//     PlcTask Outputs/GVL_iXlinker.EtherCAT_Master_ATxxxx.Beckhoff_AT1xxx.Beckhoff_AT2xxxEK1122.A_0023_AT2002_0250_0022.CC_Outputs.Control <-> CC Outputs/Control
//     PlcTask Outputs/GVL_iXlinker.EtherCAT_Master_ATxxxx.Beckhoff_AT1xxx.Beckhoff_AT2xxxEK1122.A_0023_AT2002_0250_0022.CC_Outputs.Current_setpoint_value_Ch[0] <-> CC Outputs/Current setpoint value Ch.1
//     PlcTask Outputs/GVL_iXlinker.EtherCAT_Master_ATxxxx.Beckhoff_AT1xxx.Beckhoff_AT2xxxEK1122.A_0023_AT2002_0250_0022.CC_Outputs.Current_setpoint_value_Ch[1] <-> CC Outputs/Current setpoint value Ch.2
//     PlcTask Outputs/GVL_iXlinker.EtherCAT_Master_ATxxxx.Beckhoff_AT1xxx.Beckhoff_AT2xxxEK1122.A_0023_AT2002_0250_0022.CC_Outputs.Current_setpoint_value_Ch[2] <-> CC Outputs/Current setpoint value Ch.3
//     PlcTask Outputs/GVL_iXlinker.EtherCAT_Master_ATxxxx.Beckhoff_AT1xxx.Beckhoff_AT2xxxEK1122.A_0023_AT2002_0250_0022.CC_Outputs.Current_setpoint_value_Ch[3] <-> CC Outputs/Current setpoint value Ch.4
//     PlcTask Outputs/GVL_iXlinker.EtherCAT_Master_ATxxxx.Beckhoff_AT1xxx.Beckhoff_AT2xxxEK1122.A_0023_AT2002_0250_0022.CC_Outputs.Current_setpoint_value_Ch[4] <-> CC Outputs/Current setpoint value Ch.5
//     PlcTask Outputs/GVL_iXlinker.EtherCAT_Master_ATxxxx.Beckhoff_AT1xxx.Beckhoff_AT2xxxEK1122.A_0023_AT2002_0250_0022.CC_Outputs.Current_setpoint_value_Ch[5] <-> CC Outputs/Current setpoint value Ch.6
//     PlcTask Outputs/GVL_iXlinker.EtherCAT_Master_ATxxxx.Beckhoff_AT1xxx.Beckhoff_AT2xxxEK1122.A_0023_AT2002_0250_0022.CC_Outputs.Current_setpoint_value_Ch[6] <-> CC Outputs/Current setpoint value Ch.7
//     PlcTask Outputs/GVL_iXlinker.EtherCAT_Master_ATxxxx.Beckhoff_AT1xxx.Beckhoff_AT2xxxEK1122.A_0023_AT2002_0250_0022.CC_Outputs.Current_setpoint_value_Ch[7] <-> CC Outputs/Current setpoint value Ch.8
//     PlcTask Outputs/GVL_iXlinker.EtherCAT_Master_ATxxxx.Beckhoff_AT1xxx.Beckhoff_AT2xxxEK1122.A_0023_AT2002_0250_0022.CC_Outputs.Current_setpoint_value_Ch[8] <-> CC Outputs/Current setpoint value Ch.9
//     PlcTask Outputs/GVL_iXlinker.EtherCAT_Master_ATxxxx.Beckhoff_AT1xxx.Beckhoff_AT2xxxEK1122.A_0023_AT2002_0250_0022.CC_Outputs.Current_setpoint_value_Ch[9] <-> CC Outputs/Current setpoint value Ch.10
//     PlcTask Outputs/GVL_iXlinker.EtherCAT_Master_ATxxxx.Beckhoff_AT1xxx.Beckhoff_AT2xxxEK1122.A_0023_AT2002_0250_0022.CC_Outputs.Current_setpoint_value_Ch[10] <-> CC Outputs/Current setpoint value Ch.11
//     PlcTask Outputs/GVL_iXlinker.EtherCAT_Master_ATxxxx.Beckhoff_AT1xxx.Beckhoff_AT2xxxEK1122.A_0023_AT2002_0250_0022.CC_Outputs.Current_setpoint_value_Ch[11] <-> CC Outputs/Current setpoint value Ch.12
//     PlcTask Outputs/GVL_iXlinker.EtherCAT_Master_ATxxxx.Beckhoff_AT1xxx.Beckhoff_AT2xxxEK1122.A_0023_AT2002_0250_0022.CC_Outputs.Current_setpoint_value_Ch[12] <-> CC Outputs/Current setpoint value Ch.13
//     PlcTask Outputs/GVL_iXlinker.EtherCAT_Master_ATxxxx.Beckhoff_AT1xxx.Beckhoff_AT2xxxEK1122.A_0023_AT2002_0250_0022.CC_Outputs.Current_setpoint_value_Ch[13] <-> CC Outputs/Current setpoint value Ch.14
//     PlcTask Outputs/GVL_iXlinker.EtherCAT_Master_ATxxxx.Beckhoff_AT1xxx.Beckhoff_AT2xxxEK1122.A_0023_AT2002_0250_0022.CC_Outputs.Current_setpoint_value_Ch[14] <-> CC Outputs/Current setpoint value Ch.15
//     PlcTask Inputs/GVL_iXlinker.EtherCAT_Master_ATxxxx.Beckhoff_AT1xxx.Beckhoff_AT2xxxEK1122.A_0023_AT2002_0250_0022.WcState.WcState <-> WcState/WcState
//     PlcTask Inputs/GVL_iXlinker.EtherCAT_Master_ATxxxx.Beckhoff_AT1xxx.Beckhoff_AT2xxxEK1122.A_0023_AT2002_0250_0022.WcState.InputToggle <-> WcState/InputToggle
//     PlcTask Inputs/GVL_iXlinker.EtherCAT_Master_ATxxxx.Beckhoff_AT1xxx.Beckhoff_AT2xxxEK1122.A_0023_AT2002_0250_0022.InfoData.AdsAddr <-> InfoData/AdsAddr
//     PlcTask Inputs/GVL_iXlinker.EtherCAT_Master_ATxxxx.Beckhoff_AT1xxx.Beckhoff_AT2xxxEK1122.A_0023_AT2002_0250_0022.InfoData.DcOutputShift <-> InfoData/DcOutputShift
//     PlcTask Inputs/GVL_iXlinker.EtherCAT_Master_ATxxxx.Beckhoff_AT1xxx.Beckhoff_AT2xxxEK1122.A_0023_AT2002_0250_0022.InfoData.DcInputShift <-> InfoData/DcInputShift
//     PlcTask Inputs/GVL_iXlinker.EtherCAT_Master_ATxxxx.Beckhoff_AT1xxx.Beckhoff_AT2xxxEK1122.A_0023_AT2002_0250_0022.InfoData.State <-> InfoData/State
//   PLC/PLC Instance <-> EtherCAT Master ATxxxx/Beckhoff AT1xxx/Beckhoff AT2xxxEK1122/A_0024(AT2002-0250-0023)
//     PlcTask Inputs/GVL_iXlinker.EtherCAT_Master_ATxxxx.Beckhoff_AT1xxx.Beckhoff_AT2xxxEK1122.A_0024_AT2002_0250_0023.CC_Inputs.Status <-> CC Inputs/Status
//     PlcTask Inputs/GVL_iXlinker.EtherCAT_Master_ATxxxx.Beckhoff_AT1xxx.Beckhoff_AT2xxxEK1122.A_0024_AT2002_0250_0023.CC_Inputs.Current_actual_value_Ch[0] <-> CC Inputs/Current actual value Ch.1
//     PlcTask Inputs/GVL_iXlinker.EtherCAT_Master_ATxxxx.Beckhoff_AT1xxx.Beckhoff_AT2xxxEK1122.A_0024_AT2002_0250_0023.CC_Inputs.Current_actual_value_Ch[1] <-> CC Inputs/Current actual value Ch.2
//     PlcTask Inputs/GVL_iXlinker.EtherCAT_Master_ATxxxx.Beckhoff_AT1xxx.Beckhoff_AT2xxxEK1122.A_0024_AT2002_0250_0023.CC_Inputs.Current_actual_value_Ch[2] <-> CC Inputs/Current actual value Ch.3
//     PlcTask Inputs/GVL_iXlinker.EtherCAT_Master_ATxxxx.Beckhoff_AT1xxx.Beckhoff_AT2xxxEK1122.A_0024_AT2002_0250_0023.CC_Inputs.Current_actual_value_Ch[3] <-> CC Inputs/Current actual value Ch.4
//     PlcTask Inputs/GVL_iXlinker.EtherCAT_Master_ATxxxx.Beckhoff_AT1xxx.Beckhoff_AT2xxxEK1122.A_0024_AT2002_0250_0023.CC_Inputs.Current_actual_value_Ch[4] <-> CC Inputs/Current actual value Ch.5
//     PlcTask Inputs/GVL_iXlinker.EtherCAT_Master_ATxxxx.Beckhoff_AT1xxx.Beckhoff_AT2xxxEK1122.A_0024_AT2002_0250_0023.CC_Inputs.Current_actual_value_Ch[5] <-> CC Inputs/Current actual value Ch.6
//     PlcTask Inputs/GVL_iXlinker.EtherCAT_Master_ATxxxx.Beckhoff_AT1xxx.Beckhoff_AT2xxxEK1122.A_0024_AT2002_0250_0023.CC_Inputs.Current_actual_value_Ch[6] <-> CC Inputs/Current actual value Ch.7
//     PlcTask Inputs/GVL_iXlinker.EtherCAT_Master_ATxxxx.Beckhoff_AT1xxx.Beckhoff_AT2xxxEK1122.A_0024_AT2002_0250_0023.CC_Inputs.Current_actual_value_Ch[7] <-> CC Inputs/Current actual value Ch.8
//     PlcTask Inputs/GVL_iXlinker.EtherCAT_Master_ATxxxx.Beckhoff_AT1xxx.Beckhoff_AT2xxxEK1122.A_0024_AT2002_0250_0023.CC_Inputs.Current_actual_value_Ch[8] <-> CC Inputs/Current actual value Ch.9
//     PlcTask Inputs/GVL_iXlinker.EtherCAT_Master_ATxxxx.Beckhoff_AT1xxx.Beckhoff_AT2xxxEK1122.A_0024_AT2002_0250_0023.CC_Inputs.Current_actual_value_Ch[9] <-> CC Inputs/Current actual value Ch.10
//     PlcTask Inputs/GVL_iXlinker.EtherCAT_Master_ATxxxx.Beckhoff_AT1xxx.Beckhoff_AT2xxxEK1122.A_0024_AT2002_0250_0023.CC_Inputs.Current_actual_value_Ch[10] <-> CC Inputs/Current actual value Ch.11
//     PlcTask Inputs/GVL_iXlinker.EtherCAT_Master_ATxxxx.Beckhoff_AT1xxx.Beckhoff_AT2xxxEK1122.A_0024_AT2002_0250_0023.CC_Inputs.Current_actual_value_Ch[11] <-> CC Inputs/Current actual value Ch.12
//     PlcTask Inputs/GVL_iXlinker.EtherCAT_Master_ATxxxx.Beckhoff_AT1xxx.Beckhoff_AT2xxxEK1122.A_0024_AT2002_0250_0023.CC_Inputs.Current_actual_value_Ch[12] <-> CC Inputs/Current actual value Ch.13
//     PlcTask Inputs/GVL_iXlinker.EtherCAT_Master_ATxxxx.Beckhoff_AT1xxx.Beckhoff_AT2xxxEK1122.A_0024_AT2002_0250_0023.CC_Inputs.Current_actual_value_Ch[13] <-> CC Inputs/Current actual value Ch.14
//     PlcTask Inputs/GVL_iXlinker.EtherCAT_Master_ATxxxx.Beckhoff_AT1xxx.Beckhoff_AT2xxxEK1122.A_0024_AT2002_0250_0023.CC_Inputs.Current_actual_value_Ch[14] <-> CC Inputs/Current actual value Ch.15
//     PlcTask Outputs/GVL_iXlinker.EtherCAT_Master_ATxxxx.Beckhoff_AT1xxx.Beckhoff_AT2xxxEK1122.A_0024_AT2002_0250_0023.CC_Outputs.Control <-> CC Outputs/Control
//     PlcTask Outputs/GVL_iXlinker.EtherCAT_Master_ATxxxx.Beckhoff_AT1xxx.Beckhoff_AT2xxxEK1122.A_0024_AT2002_0250_0023.CC_Outputs.Current_setpoint_value_Ch[0] <-> CC Outputs/Current setpoint value Ch.1
//     PlcTask Outputs/GVL_iXlinker.EtherCAT_Master_ATxxxx.Beckhoff_AT1xxx.Beckhoff_AT2xxxEK1122.A_0024_AT2002_0250_0023.CC_Outputs.Current_setpoint_value_Ch[1] <-> CC Outputs/Current setpoint value Ch.2
//     PlcTask Outputs/GVL_iXlinker.EtherCAT_Master_ATxxxx.Beckhoff_AT1xxx.Beckhoff_AT2xxxEK1122.A_0024_AT2002_0250_0023.CC_Outputs.Current_setpoint_value_Ch[2] <-> CC Outputs/Current setpoint value Ch.3
//     PlcTask Outputs/GVL_iXlinker.EtherCAT_Master_ATxxxx.Beckhoff_AT1xxx.Beckhoff_AT2xxxEK1122.A_0024_AT2002_0250_0023.CC_Outputs.Current_setpoint_value_Ch[3] <-> CC Outputs/Current setpoint value Ch.4
//     PlcTask Outputs/GVL_iXlinker.EtherCAT_Master_ATxxxx.Beckhoff_AT1xxx.Beckhoff_AT2xxxEK1122.A_0024_AT2002_0250_0023.CC_Outputs.Current_setpoint_value_Ch[4] <-> CC Outputs/Current setpoint value Ch.5
//     PlcTask Outputs/GVL_iXlinker.EtherCAT_Master_ATxxxx.Beckhoff_AT1xxx.Beckhoff_AT2xxxEK1122.A_0024_AT2002_0250_0023.CC_Outputs.Current_setpoint_value_Ch[5] <-> CC Outputs/Current setpoint value Ch.6
//     PlcTask Outputs/GVL_iXlinker.EtherCAT_Master_ATxxxx.Beckhoff_AT1xxx.Beckhoff_AT2xxxEK1122.A_0024_AT2002_0250_0023.CC_Outputs.Current_setpoint_value_Ch[6] <-> CC Outputs/Current setpoint value Ch.7
//     PlcTask Outputs/GVL_iXlinker.EtherCAT_Master_ATxxxx.Beckhoff_AT1xxx.Beckhoff_AT2xxxEK1122.A_0024_AT2002_0250_0023.CC_Outputs.Current_setpoint_value_Ch[7] <-> CC Outputs/Current setpoint value Ch.8
//     PlcTask Outputs/GVL_iXlinker.EtherCAT_Master_ATxxxx.Beckhoff_AT1xxx.Beckhoff_AT2xxxEK1122.A_0024_AT2002_0250_0023.CC_Outputs.Current_setpoint_value_Ch[8] <-> CC Outputs/Current setpoint value Ch.9
//     PlcTask Outputs/GVL_iXlinker.EtherCAT_Master_ATxxxx.Beckhoff_AT1xxx.Beckhoff_AT2xxxEK1122.A_0024_AT2002_0250_0023.CC_Outputs.Current_setpoint_value_Ch[9] <-> CC Outputs/Current setpoint value Ch.10
//     PlcTask Outputs/GVL_iXlinker.EtherCAT_Master_ATxxxx.Beckhoff_AT1xxx.Beckhoff_AT2xxxEK1122.A_0024_AT2002_0250_0023.CC_Outputs.Current_setpoint_value_Ch[10] <-> CC Outputs/Current setpoint value Ch.11
//     PlcTask Outputs/GVL_iXlinker.EtherCAT_Master_ATxxxx.Beckhoff_AT1xxx.Beckhoff_AT2xxxEK1122.A_0024_AT2002_0250_0023.CC_Outputs.Current_setpoint_value_Ch[11] <-> CC Outputs/Current setpoint value Ch.12
//     PlcTask Outputs/GVL_iXlinker.EtherCAT_Master_ATxxxx.Beckhoff_AT1xxx.Beckhoff_AT2xxxEK1122.A_0024_AT2002_0250_0023.CC_Outputs.Current_setpoint_value_Ch[12] <-> CC Outputs/Current setpoint value Ch.13
//     PlcTask Outputs/GVL_iXlinker.EtherCAT_Master_ATxxxx.Beckhoff_AT1xxx.Beckhoff_AT2xxxEK1122.A_0024_AT2002_0250_0023.CC_Outputs.Current_setpoint_value_Ch[13] <-> CC Outputs/Current setpoint value Ch.14
//     PlcTask Outputs/GVL_iXlinker.EtherCAT_Master_ATxxxx.Beckhoff_AT1xxx.Beckhoff_AT2xxxEK1122.A_0024_AT2002_0250_0023.CC_Outputs.Current_setpoint_value_Ch[14] <-> CC Outputs/Current setpoint value Ch.15
//     PlcTask Inputs/GVL_iXlinker.EtherCAT_Master_ATxxxx.Beckhoff_AT1xxx.Beckhoff_AT2xxxEK1122.A_0024_AT2002_0250_0023.WcState.WcState <-> WcState/WcState
//     PlcTask Inputs/GVL_iXlinker.EtherCAT_Master_ATxxxx.Beckhoff_AT1xxx.Beckhoff_AT2xxxEK1122.A_0024_AT2002_0250_0023.WcState.InputToggle <-> WcState/InputToggle
//     PlcTask Inputs/GVL_iXlinker.EtherCAT_Master_ATxxxx.Beckhoff_AT1xxx.Beckhoff_AT2xxxEK1122.A_0024_AT2002_0250_0023.InfoData.AdsAddr <-> InfoData/AdsAddr
//     PlcTask Inputs/GVL_iXlinker.EtherCAT_Master_ATxxxx.Beckhoff_AT1xxx.Beckhoff_AT2xxxEK1122.A_0024_AT2002_0250_0023.InfoData.DcOutputShift <-> InfoData/DcOutputShift
//     PlcTask Inputs/GVL_iXlinker.EtherCAT_Master_ATxxxx.Beckhoff_AT1xxx.Beckhoff_AT2xxxEK1122.A_0024_AT2002_0250_0023.InfoData.DcInputShift <-> InfoData/DcInputShift
//     PlcTask Inputs/GVL_iXlinker.EtherCAT_Master_ATxxxx.Beckhoff_AT1xxx.Beckhoff_AT2xxxEK1122.A_0024_AT2002_0250_0023.InfoData.State <-> InfoData/State
//   PLC/PLC Instance <-> EtherCAT Master ATxxxx/Beckhoff AT1xxx/Beckhoff AT2xxxEK1122/A_0025(AT2002-0250-0024)
//     PlcTask Inputs/GVL_iXlinker.EtherCAT_Master_ATxxxx.Beckhoff_AT1xxx.Beckhoff_AT2xxxEK1122.A_0025_AT2002_0250_0024.CC_Inputs.Status <-> CC Inputs/Status
//     PlcTask Inputs/GVL_iXlinker.EtherCAT_Master_ATxxxx.Beckhoff_AT1xxx.Beckhoff_AT2xxxEK1122.A_0025_AT2002_0250_0024.CC_Inputs.Current_actual_value_Ch[0] <-> CC Inputs/Current actual value Ch.1
//     PlcTask Inputs/GVL_iXlinker.EtherCAT_Master_ATxxxx.Beckhoff_AT1xxx.Beckhoff_AT2xxxEK1122.A_0025_AT2002_0250_0024.CC_Inputs.Current_actual_value_Ch[1] <-> CC Inputs/Current actual value Ch.2
//     PlcTask Inputs/GVL_iXlinker.EtherCAT_Master_ATxxxx.Beckhoff_AT1xxx.Beckhoff_AT2xxxEK1122.A_0025_AT2002_0250_0024.CC_Inputs.Current_actual_value_Ch[2] <-> CC Inputs/Current actual value Ch.3
//     PlcTask Inputs/GVL_iXlinker.EtherCAT_Master_ATxxxx.Beckhoff_AT1xxx.Beckhoff_AT2xxxEK1122.A_0025_AT2002_0250_0024.CC_Inputs.Current_actual_value_Ch[3] <-> CC Inputs/Current actual value Ch.4
//     PlcTask Inputs/GVL_iXlinker.EtherCAT_Master_ATxxxx.Beckhoff_AT1xxx.Beckhoff_AT2xxxEK1122.A_0025_AT2002_0250_0024.CC_Inputs.Current_actual_value_Ch[4] <-> CC Inputs/Current actual value Ch.5
//     PlcTask Inputs/GVL_iXlinker.EtherCAT_Master_ATxxxx.Beckhoff_AT1xxx.Beckhoff_AT2xxxEK1122.A_0025_AT2002_0250_0024.CC_Inputs.Current_actual_value_Ch[5] <-> CC Inputs/Current actual value Ch.6
//     PlcTask Inputs/GVL_iXlinker.EtherCAT_Master_ATxxxx.Beckhoff_AT1xxx.Beckhoff_AT2xxxEK1122.A_0025_AT2002_0250_0024.CC_Inputs.Current_actual_value_Ch[6] <-> CC Inputs/Current actual value Ch.7
//     PlcTask Inputs/GVL_iXlinker.EtherCAT_Master_ATxxxx.Beckhoff_AT1xxx.Beckhoff_AT2xxxEK1122.A_0025_AT2002_0250_0024.CC_Inputs.Current_actual_value_Ch[7] <-> CC Inputs/Current actual value Ch.8
//     PlcTask Inputs/GVL_iXlinker.EtherCAT_Master_ATxxxx.Beckhoff_AT1xxx.Beckhoff_AT2xxxEK1122.A_0025_AT2002_0250_0024.CC_Inputs.Current_actual_value_Ch[8] <-> CC Inputs/Current actual value Ch.9
//     PlcTask Inputs/GVL_iXlinker.EtherCAT_Master_ATxxxx.Beckhoff_AT1xxx.Beckhoff_AT2xxxEK1122.A_0025_AT2002_0250_0024.CC_Inputs.Current_actual_value_Ch[9] <-> CC Inputs/Current actual value Ch.10
//     PlcTask Inputs/GVL_iXlinker.EtherCAT_Master_ATxxxx.Beckhoff_AT1xxx.Beckhoff_AT2xxxEK1122.A_0025_AT2002_0250_0024.CC_Inputs.Current_actual_value_Ch[10] <-> CC Inputs/Current actual value Ch.11
//     PlcTask Inputs/GVL_iXlinker.EtherCAT_Master_ATxxxx.Beckhoff_AT1xxx.Beckhoff_AT2xxxEK1122.A_0025_AT2002_0250_0024.CC_Inputs.Current_actual_value_Ch[11] <-> CC Inputs/Current actual value Ch.12
//     PlcTask Inputs/GVL_iXlinker.EtherCAT_Master_ATxxxx.Beckhoff_AT1xxx.Beckhoff_AT2xxxEK1122.A_0025_AT2002_0250_0024.CC_Inputs.Current_actual_value_Ch[12] <-> CC Inputs/Current actual value Ch.13
//     PlcTask Inputs/GVL_iXlinker.EtherCAT_Master_ATxxxx.Beckhoff_AT1xxx.Beckhoff_AT2xxxEK1122.A_0025_AT2002_0250_0024.CC_Inputs.Current_actual_value_Ch[13] <-> CC Inputs/Current actual value Ch.14
//     PlcTask Inputs/GVL_iXlinker.EtherCAT_Master_ATxxxx.Beckhoff_AT1xxx.Beckhoff_AT2xxxEK1122.A_0025_AT2002_0250_0024.CC_Inputs.Current_actual_value_Ch[14] <-> CC Inputs/Current actual value Ch.15
//     PlcTask Outputs/GVL_iXlinker.EtherCAT_Master_ATxxxx.Beckhoff_AT1xxx.Beckhoff_AT2xxxEK1122.A_0025_AT2002_0250_0024.CC_Outputs.Control <-> CC Outputs/Control
//     PlcTask Outputs/GVL_iXlinker.EtherCAT_Master_ATxxxx.Beckhoff_AT1xxx.Beckhoff_AT2xxxEK1122.A_0025_AT2002_0250_0024.CC_Outputs.Current_setpoint_value_Ch[0] <-> CC Outputs/Current setpoint value Ch.1
//     PlcTask Outputs/GVL_iXlinker.EtherCAT_Master_ATxxxx.Beckhoff_AT1xxx.Beckhoff_AT2xxxEK1122.A_0025_AT2002_0250_0024.CC_Outputs.Current_setpoint_value_Ch[1] <-> CC Outputs/Current setpoint value Ch.2
//     PlcTask Outputs/GVL_iXlinker.EtherCAT_Master_ATxxxx.Beckhoff_AT1xxx.Beckhoff_AT2xxxEK1122.A_0025_AT2002_0250_0024.CC_Outputs.Current_setpoint_value_Ch[2] <-> CC Outputs/Current setpoint value Ch.3
//     PlcTask Outputs/GVL_iXlinker.EtherCAT_Master_ATxxxx.Beckhoff_AT1xxx.Beckhoff_AT2xxxEK1122.A_0025_AT2002_0250_0024.CC_Outputs.Current_setpoint_value_Ch[3] <-> CC Outputs/Current setpoint value Ch.4
//     PlcTask Outputs/GVL_iXlinker.EtherCAT_Master_ATxxxx.Beckhoff_AT1xxx.Beckhoff_AT2xxxEK1122.A_0025_AT2002_0250_0024.CC_Outputs.Current_setpoint_value_Ch[4] <-> CC Outputs/Current setpoint value Ch.5
//     PlcTask Outputs/GVL_iXlinker.EtherCAT_Master_ATxxxx.Beckhoff_AT1xxx.Beckhoff_AT2xxxEK1122.A_0025_AT2002_0250_0024.CC_Outputs.Current_setpoint_value_Ch[5] <-> CC Outputs/Current setpoint value Ch.6
//     PlcTask Outputs/GVL_iXlinker.EtherCAT_Master_ATxxxx.Beckhoff_AT1xxx.Beckhoff_AT2xxxEK1122.A_0025_AT2002_0250_0024.CC_Outputs.Current_setpoint_value_Ch[6] <-> CC Outputs/Current setpoint value Ch.7
//     PlcTask Outputs/GVL_iXlinker.EtherCAT_Master_ATxxxx.Beckhoff_AT1xxx.Beckhoff_AT2xxxEK1122.A_0025_AT2002_0250_0024.CC_Outputs.Current_setpoint_value_Ch[7] <-> CC Outputs/Current setpoint value Ch.8
//     PlcTask Outputs/GVL_iXlinker.EtherCAT_Master_ATxxxx.Beckhoff_AT1xxx.Beckhoff_AT2xxxEK1122.A_0025_AT2002_0250_0024.CC_Outputs.Current_setpoint_value_Ch[8] <-> CC Outputs/Current setpoint value Ch.9
//     PlcTask Outputs/GVL_iXlinker.EtherCAT_Master_ATxxxx.Beckhoff_AT1xxx.Beckhoff_AT2xxxEK1122.A_0025_AT2002_0250_0024.CC_Outputs.Current_setpoint_value_Ch[9] <-> CC Outputs/Current setpoint value Ch.10
//     PlcTask Outputs/GVL_iXlinker.EtherCAT_Master_ATxxxx.Beckhoff_AT1xxx.Beckhoff_AT2xxxEK1122.A_0025_AT2002_0250_0024.CC_Outputs.Current_setpoint_value_Ch[10] <-> CC Outputs/Current setpoint value Ch.11
//     PlcTask Outputs/GVL_iXlinker.EtherCAT_Master_ATxxxx.Beckhoff_AT1xxx.Beckhoff_AT2xxxEK1122.A_0025_AT2002_0250_0024.CC_Outputs.Current_setpoint_value_Ch[11] <-> CC Outputs/Current setpoint value Ch.12
//     PlcTask Outputs/GVL_iXlinker.EtherCAT_Master_ATxxxx.Beckhoff_AT1xxx.Beckhoff_AT2xxxEK1122.A_0025_AT2002_0250_0024.CC_Outputs.Current_setpoint_value_Ch[12] <-> CC Outputs/Current setpoint value Ch.13
//     PlcTask Outputs/GVL_iXlinker.EtherCAT_Master_ATxxxx.Beckhoff_AT1xxx.Beckhoff_AT2xxxEK1122.A_0025_AT2002_0250_0024.CC_Outputs.Current_setpoint_value_Ch[13] <-> CC Outputs/Current setpoint value Ch.14
//     PlcTask Outputs/GVL_iXlinker.EtherCAT_Master_ATxxxx.Beckhoff_AT1xxx.Beckhoff_AT2xxxEK1122.A_0025_AT2002_0250_0024.CC_Outputs.Current_setpoint_value_Ch[14] <-> CC Outputs/Current setpoint value Ch.15
//     PlcTask Inputs/GVL_iXlinker.EtherCAT_Master_ATxxxx.Beckhoff_AT1xxx.Beckhoff_AT2xxxEK1122.A_0025_AT2002_0250_0024.WcState.WcState <-> WcState/WcState
//     PlcTask Inputs/GVL_iXlinker.EtherCAT_Master_ATxxxx.Beckhoff_AT1xxx.Beckhoff_AT2xxxEK1122.A_0025_AT2002_0250_0024.WcState.InputToggle <-> WcState/InputToggle
//     PlcTask Inputs/GVL_iXlinker.EtherCAT_Master_ATxxxx.Beckhoff_AT1xxx.Beckhoff_AT2xxxEK1122.A_0025_AT2002_0250_0024.InfoData.AdsAddr <-> InfoData/AdsAddr
//     PlcTask Inputs/GVL_iXlinker.EtherCAT_Master_ATxxxx.Beckhoff_AT1xxx.Beckhoff_AT2xxxEK1122.A_0025_AT2002_0250_0024.InfoData.DcOutputShift <-> InfoData/DcOutputShift
//     PlcTask Inputs/GVL_iXlinker.EtherCAT_Master_ATxxxx.Beckhoff_AT1xxx.Beckhoff_AT2xxxEK1122.A_0025_AT2002_0250_0024.InfoData.DcInputShift <-> InfoData/DcInputShift
//     PlcTask Inputs/GVL_iXlinker.EtherCAT_Master_ATxxxx.Beckhoff_AT1xxx.Beckhoff_AT2xxxEK1122.A_0025_AT2002_0250_0024.InfoData.State <-> InfoData/State
//   PLC/PLC Instance <-> EtherCAT Master ATxxxx/Beckhoff AT1xxx/Beckhoff AT2xxxEK1122/A_0026(AT2020-0250-0018)
//     PlcTask Inputs/GVL_iXlinker.EtherCAT_Master_ATxxxx.Beckhoff_AT1xxx.Beckhoff_AT2xxxEK1122.A_0026_AT2020_0250_0018.CC_Inputs.Status <-> CC Inputs/Status
//     PlcTask Inputs/GVL_iXlinker.EtherCAT_Master_ATxxxx.Beckhoff_AT1xxx.Beckhoff_AT2xxxEK1122.A_0026_AT2020_0250_0018.CC_Inputs.Current_actual_value_Ch[0] <-> CC Inputs/Current actual value Ch.1
//     PlcTask Inputs/GVL_iXlinker.EtherCAT_Master_ATxxxx.Beckhoff_AT1xxx.Beckhoff_AT2xxxEK1122.A_0026_AT2020_0250_0018.CC_Inputs.Current_actual_value_Ch[1] <-> CC Inputs/Current actual value Ch.2
//     PlcTask Inputs/GVL_iXlinker.EtherCAT_Master_ATxxxx.Beckhoff_AT1xxx.Beckhoff_AT2xxxEK1122.A_0026_AT2020_0250_0018.CC_Inputs.Current_actual_value_Ch[2] <-> CC Inputs/Current actual value Ch.3
//     PlcTask Inputs/GVL_iXlinker.EtherCAT_Master_ATxxxx.Beckhoff_AT1xxx.Beckhoff_AT2xxxEK1122.A_0026_AT2020_0250_0018.CC_Inputs.Current_actual_value_Ch[3] <-> CC Inputs/Current actual value Ch.4
//     PlcTask Inputs/GVL_iXlinker.EtherCAT_Master_ATxxxx.Beckhoff_AT1xxx.Beckhoff_AT2xxxEK1122.A_0026_AT2020_0250_0018.CC_Inputs.Current_actual_value_Ch[4] <-> CC Inputs/Current actual value Ch.5
//     PlcTask Inputs/GVL_iXlinker.EtherCAT_Master_ATxxxx.Beckhoff_AT1xxx.Beckhoff_AT2xxxEK1122.A_0026_AT2020_0250_0018.CC_Inputs.Current_actual_value_Ch[5] <-> CC Inputs/Current actual value Ch.6
//     PlcTask Inputs/GVL_iXlinker.EtherCAT_Master_ATxxxx.Beckhoff_AT1xxx.Beckhoff_AT2xxxEK1122.A_0026_AT2020_0250_0018.CC_Inputs.Current_actual_value_Ch[6] <-> CC Inputs/Current actual value Ch.7
//     PlcTask Inputs/GVL_iXlinker.EtherCAT_Master_ATxxxx.Beckhoff_AT1xxx.Beckhoff_AT2xxxEK1122.A_0026_AT2020_0250_0018.CC_Inputs.Current_actual_value_Ch[7] <-> CC Inputs/Current actual value Ch.8
//     PlcTask Inputs/GVL_iXlinker.EtherCAT_Master_ATxxxx.Beckhoff_AT1xxx.Beckhoff_AT2xxxEK1122.A_0026_AT2020_0250_0018.CC_Inputs.Current_actual_value_Ch[8] <-> CC Inputs/Current actual value Ch.9
//     PlcTask Inputs/GVL_iXlinker.EtherCAT_Master_ATxxxx.Beckhoff_AT1xxx.Beckhoff_AT2xxxEK1122.A_0026_AT2020_0250_0018.CC_Inputs.Current_actual_value_Ch[9] <-> CC Inputs/Current actual value Ch.10
//     PlcTask Inputs/GVL_iXlinker.EtherCAT_Master_ATxxxx.Beckhoff_AT1xxx.Beckhoff_AT2xxxEK1122.A_0026_AT2020_0250_0018.CC_Inputs.Current_actual_value_Ch[10] <-> CC Inputs/Current actual value Ch.11
//     PlcTask Inputs/GVL_iXlinker.EtherCAT_Master_ATxxxx.Beckhoff_AT1xxx.Beckhoff_AT2xxxEK1122.A_0026_AT2020_0250_0018.CC_Inputs.Current_actual_value_Ch[11] <-> CC Inputs/Current actual value Ch.12
//     PlcTask Inputs/GVL_iXlinker.EtherCAT_Master_ATxxxx.Beckhoff_AT1xxx.Beckhoff_AT2xxxEK1122.A_0026_AT2020_0250_0018.CC_Inputs.Current_actual_value_Ch[12] <-> CC Inputs/Current actual value Ch.13
//     PlcTask Inputs/GVL_iXlinker.EtherCAT_Master_ATxxxx.Beckhoff_AT1xxx.Beckhoff_AT2xxxEK1122.A_0026_AT2020_0250_0018.CC_Inputs.Current_actual_value_Ch[13] <-> CC Inputs/Current actual value Ch.14
//     PlcTask Inputs/GVL_iXlinker.EtherCAT_Master_ATxxxx.Beckhoff_AT1xxx.Beckhoff_AT2xxxEK1122.A_0026_AT2020_0250_0018.CC_Inputs.Current_actual_value_Ch[14] <-> CC Inputs/Current actual value Ch.15
//     PlcTask Outputs/GVL_iXlinker.EtherCAT_Master_ATxxxx.Beckhoff_AT1xxx.Beckhoff_AT2xxxEK1122.A_0026_AT2020_0250_0018.CC_Outputs.Control <-> CC Outputs/Control
//     PlcTask Outputs/GVL_iXlinker.EtherCAT_Master_ATxxxx.Beckhoff_AT1xxx.Beckhoff_AT2xxxEK1122.A_0026_AT2020_0250_0018.CC_Outputs.Current_setpoint_value_Ch[0] <-> CC Outputs/Current setpoint value Ch.1
//     PlcTask Outputs/GVL_iXlinker.EtherCAT_Master_ATxxxx.Beckhoff_AT1xxx.Beckhoff_AT2xxxEK1122.A_0026_AT2020_0250_0018.CC_Outputs.Current_setpoint_value_Ch[1] <-> CC Outputs/Current setpoint value Ch.2
//     PlcTask Outputs/GVL_iXlinker.EtherCAT_Master_ATxxxx.Beckhoff_AT1xxx.Beckhoff_AT2xxxEK1122.A_0026_AT2020_0250_0018.CC_Outputs.Current_setpoint_value_Ch[2] <-> CC Outputs/Current setpoint value Ch.3
//     PlcTask Outputs/GVL_iXlinker.EtherCAT_Master_ATxxxx.Beckhoff_AT1xxx.Beckhoff_AT2xxxEK1122.A_0026_AT2020_0250_0018.CC_Outputs.Current_setpoint_value_Ch[3] <-> CC Outputs/Current setpoint value Ch.4
//     PlcTask Outputs/GVL_iXlinker.EtherCAT_Master_ATxxxx.Beckhoff_AT1xxx.Beckhoff_AT2xxxEK1122.A_0026_AT2020_0250_0018.CC_Outputs.Current_setpoint_value_Ch[4] <-> CC Outputs/Current setpoint value Ch.5
//     PlcTask Outputs/GVL_iXlinker.EtherCAT_Master_ATxxxx.Beckhoff_AT1xxx.Beckhoff_AT2xxxEK1122.A_0026_AT2020_0250_0018.CC_Outputs.Current_setpoint_value_Ch[5] <-> CC Outputs/Current setpoint value Ch.6
//     PlcTask Outputs/GVL_iXlinker.EtherCAT_Master_ATxxxx.Beckhoff_AT1xxx.Beckhoff_AT2xxxEK1122.A_0026_AT2020_0250_0018.CC_Outputs.Current_setpoint_value_Ch[6] <-> CC Outputs/Current setpoint value Ch.7
//     PlcTask Outputs/GVL_iXlinker.EtherCAT_Master_ATxxxx.Beckhoff_AT1xxx.Beckhoff_AT2xxxEK1122.A_0026_AT2020_0250_0018.CC_Outputs.Current_setpoint_value_Ch[7] <-> CC Outputs/Current setpoint value Ch.8
//     PlcTask Outputs/GVL_iXlinker.EtherCAT_Master_ATxxxx.Beckhoff_AT1xxx.Beckhoff_AT2xxxEK1122.A_0026_AT2020_0250_0018.CC_Outputs.Current_setpoint_value_Ch[8] <-> CC Outputs/Current setpoint value Ch.9
//     PlcTask Outputs/GVL_iXlinker.EtherCAT_Master_ATxxxx.Beckhoff_AT1xxx.Beckhoff_AT2xxxEK1122.A_0026_AT2020_0250_0018.CC_Outputs.Current_setpoint_value_Ch[9] <-> CC Outputs/Current setpoint value Ch.10
//     PlcTask Outputs/GVL_iXlinker.EtherCAT_Master_ATxxxx.Beckhoff_AT1xxx.Beckhoff_AT2xxxEK1122.A_0026_AT2020_0250_0018.CC_Outputs.Current_setpoint_value_Ch[10] <-> CC Outputs/Current setpoint value Ch.11
//     PlcTask Outputs/GVL_iXlinker.EtherCAT_Master_ATxxxx.Beckhoff_AT1xxx.Beckhoff_AT2xxxEK1122.A_0026_AT2020_0250_0018.CC_Outputs.Current_setpoint_value_Ch[11] <-> CC Outputs/Current setpoint value Ch.12
//     PlcTask Outputs/GVL_iXlinker.EtherCAT_Master_ATxxxx.Beckhoff_AT1xxx.Beckhoff_AT2xxxEK1122.A_0026_AT2020_0250_0018.CC_Outputs.Current_setpoint_value_Ch[12] <-> CC Outputs/Current setpoint value Ch.13
//     PlcTask Outputs/GVL_iXlinker.EtherCAT_Master_ATxxxx.Beckhoff_AT1xxx.Beckhoff_AT2xxxEK1122.A_0026_AT2020_0250_0018.CC_Outputs.Current_setpoint_value_Ch[13] <-> CC Outputs/Current setpoint value Ch.14
//     PlcTask Outputs/GVL_iXlinker.EtherCAT_Master_ATxxxx.Beckhoff_AT1xxx.Beckhoff_AT2xxxEK1122.A_0026_AT2020_0250_0018.CC_Outputs.Current_setpoint_value_Ch[14] <-> CC Outputs/Current setpoint value Ch.15
//     PlcTask Inputs/GVL_iXlinker.EtherCAT_Master_ATxxxx.Beckhoff_AT1xxx.Beckhoff_AT2xxxEK1122.A_0026_AT2020_0250_0018.WcState.WcState <-> WcState/WcState
//     PlcTask Inputs/GVL_iXlinker.EtherCAT_Master_ATxxxx.Beckhoff_AT1xxx.Beckhoff_AT2xxxEK1122.A_0026_AT2020_0250_0018.WcState.InputToggle <-> WcState/InputToggle
//     PlcTask Inputs/GVL_iXlinker.EtherCAT_Master_ATxxxx.Beckhoff_AT1xxx.Beckhoff_AT2xxxEK1122.A_0026_AT2020_0250_0018.InfoData.AdsAddr <-> InfoData/AdsAddr
//     PlcTask Inputs/GVL_iXlinker.EtherCAT_Master_ATxxxx.Beckhoff_AT1xxx.Beckhoff_AT2xxxEK1122.A_0026_AT2020_0250_0018.InfoData.DcOutputShift <-> InfoData/DcOutputShift
//     PlcTask Inputs/GVL_iXlinker.EtherCAT_Master_ATxxxx.Beckhoff_AT1xxx.Beckhoff_AT2xxxEK1122.A_0026_AT2020_0250_0018.InfoData.DcInputShift <-> InfoData/DcInputShift
//     PlcTask Inputs/GVL_iXlinker.EtherCAT_Master_ATxxxx.Beckhoff_AT1xxx.Beckhoff_AT2xxxEK1122.A_0026_AT2020_0250_0018.InfoData.State <-> InfoData/State
//   PLC/PLC Instance <-> EtherCAT Master ATxxxx/Beckhoff AT1xxx/Beckhoff AT2xxxEK1122/A_0027(AT2020-0250-0021)
//     PlcTask Inputs/GVL_iXlinker.EtherCAT_Master_ATxxxx.Beckhoff_AT1xxx.Beckhoff_AT2xxxEK1122.A_0027_AT2020_0250_0021.CC_Inputs.Status <-> CC Inputs/Status
//     PlcTask Inputs/GVL_iXlinker.EtherCAT_Master_ATxxxx.Beckhoff_AT1xxx.Beckhoff_AT2xxxEK1122.A_0027_AT2020_0250_0021.CC_Inputs.Current_actual_value_Ch[0] <-> CC Inputs/Current actual value Ch.1
//     PlcTask Inputs/GVL_iXlinker.EtherCAT_Master_ATxxxx.Beckhoff_AT1xxx.Beckhoff_AT2xxxEK1122.A_0027_AT2020_0250_0021.CC_Inputs.Current_actual_value_Ch[1] <-> CC Inputs/Current actual value Ch.2
//     PlcTask Inputs/GVL_iXlinker.EtherCAT_Master_ATxxxx.Beckhoff_AT1xxx.Beckhoff_AT2xxxEK1122.A_0027_AT2020_0250_0021.CC_Inputs.Current_actual_value_Ch[2] <-> CC Inputs/Current actual value Ch.3
//     PlcTask Inputs/GVL_iXlinker.EtherCAT_Master_ATxxxx.Beckhoff_AT1xxx.Beckhoff_AT2xxxEK1122.A_0027_AT2020_0250_0021.CC_Inputs.Current_actual_value_Ch[3] <-> CC Inputs/Current actual value Ch.4
//     PlcTask Inputs/GVL_iXlinker.EtherCAT_Master_ATxxxx.Beckhoff_AT1xxx.Beckhoff_AT2xxxEK1122.A_0027_AT2020_0250_0021.CC_Inputs.Current_actual_value_Ch[4] <-> CC Inputs/Current actual value Ch.5
//     PlcTask Inputs/GVL_iXlinker.EtherCAT_Master_ATxxxx.Beckhoff_AT1xxx.Beckhoff_AT2xxxEK1122.A_0027_AT2020_0250_0021.CC_Inputs.Current_actual_value_Ch[5] <-> CC Inputs/Current actual value Ch.6
//     PlcTask Inputs/GVL_iXlinker.EtherCAT_Master_ATxxxx.Beckhoff_AT1xxx.Beckhoff_AT2xxxEK1122.A_0027_AT2020_0250_0021.CC_Inputs.Current_actual_value_Ch[6] <-> CC Inputs/Current actual value Ch.7
//     PlcTask Inputs/GVL_iXlinker.EtherCAT_Master_ATxxxx.Beckhoff_AT1xxx.Beckhoff_AT2xxxEK1122.A_0027_AT2020_0250_0021.CC_Inputs.Current_actual_value_Ch[7] <-> CC Inputs/Current actual value Ch.8
//     PlcTask Inputs/GVL_iXlinker.EtherCAT_Master_ATxxxx.Beckhoff_AT1xxx.Beckhoff_AT2xxxEK1122.A_0027_AT2020_0250_0021.CC_Inputs.Current_actual_value_Ch[8] <-> CC Inputs/Current actual value Ch.9
//     PlcTask Inputs/GVL_iXlinker.EtherCAT_Master_ATxxxx.Beckhoff_AT1xxx.Beckhoff_AT2xxxEK1122.A_0027_AT2020_0250_0021.CC_Inputs.Current_actual_value_Ch[9] <-> CC Inputs/Current actual value Ch.10
//     PlcTask Inputs/GVL_iXlinker.EtherCAT_Master_ATxxxx.Beckhoff_AT1xxx.Beckhoff_AT2xxxEK1122.A_0027_AT2020_0250_0021.CC_Inputs.Current_actual_value_Ch[10] <-> CC Inputs/Current actual value Ch.11
//     PlcTask Inputs/GVL_iXlinker.EtherCAT_Master_ATxxxx.Beckhoff_AT1xxx.Beckhoff_AT2xxxEK1122.A_0027_AT2020_0250_0021.CC_Inputs.Current_actual_value_Ch[11] <-> CC Inputs/Current actual value Ch.12
//     PlcTask Inputs/GVL_iXlinker.EtherCAT_Master_ATxxxx.Beckhoff_AT1xxx.Beckhoff_AT2xxxEK1122.A_0027_AT2020_0250_0021.CC_Inputs.Current_actual_value_Ch[12] <-> CC Inputs/Current actual value Ch.13
//     PlcTask Inputs/GVL_iXlinker.EtherCAT_Master_ATxxxx.Beckhoff_AT1xxx.Beckhoff_AT2xxxEK1122.A_0027_AT2020_0250_0021.CC_Inputs.Current_actual_value_Ch[13] <-> CC Inputs/Current actual value Ch.14
//     PlcTask Inputs/GVL_iXlinker.EtherCAT_Master_ATxxxx.Beckhoff_AT1xxx.Beckhoff_AT2xxxEK1122.A_0027_AT2020_0250_0021.CC_Inputs.Current_actual_value_Ch[14] <-> CC Inputs/Current actual value Ch.15
//     PlcTask Outputs/GVL_iXlinker.EtherCAT_Master_ATxxxx.Beckhoff_AT1xxx.Beckhoff_AT2xxxEK1122.A_0027_AT2020_0250_0021.CC_Outputs.Control <-> CC Outputs/Control
//     PlcTask Outputs/GVL_iXlinker.EtherCAT_Master_ATxxxx.Beckhoff_AT1xxx.Beckhoff_AT2xxxEK1122.A_0027_AT2020_0250_0021.CC_Outputs.Current_setpoint_value_Ch[0] <-> CC Outputs/Current setpoint value Ch.1
//     PlcTask Outputs/GVL_iXlinker.EtherCAT_Master_ATxxxx.Beckhoff_AT1xxx.Beckhoff_AT2xxxEK1122.A_0027_AT2020_0250_0021.CC_Outputs.Current_setpoint_value_Ch[1] <-> CC Outputs/Current setpoint value Ch.2
//     PlcTask Outputs/GVL_iXlinker.EtherCAT_Master_ATxxxx.Beckhoff_AT1xxx.Beckhoff_AT2xxxEK1122.A_0027_AT2020_0250_0021.CC_Outputs.Current_setpoint_value_Ch[2] <-> CC Outputs/Current setpoint value Ch.3
//     PlcTask Outputs/GVL_iXlinker.EtherCAT_Master_ATxxxx.Beckhoff_AT1xxx.Beckhoff_AT2xxxEK1122.A_0027_AT2020_0250_0021.CC_Outputs.Current_setpoint_value_Ch[3] <-> CC Outputs/Current setpoint value Ch.4
//     PlcTask Outputs/GVL_iXlinker.EtherCAT_Master_ATxxxx.Beckhoff_AT1xxx.Beckhoff_AT2xxxEK1122.A_0027_AT2020_0250_0021.CC_Outputs.Current_setpoint_value_Ch[4] <-> CC Outputs/Current setpoint value Ch.5
//     PlcTask Outputs/GVL_iXlinker.EtherCAT_Master_ATxxxx.Beckhoff_AT1xxx.Beckhoff_AT2xxxEK1122.A_0027_AT2020_0250_0021.CC_Outputs.Current_setpoint_value_Ch[5] <-> CC Outputs/Current setpoint value Ch.6
//     PlcTask Outputs/GVL_iXlinker.EtherCAT_Master_ATxxxx.Beckhoff_AT1xxx.Beckhoff_AT2xxxEK1122.A_0027_AT2020_0250_0021.CC_Outputs.Current_setpoint_value_Ch[6] <-> CC Outputs/Current setpoint value Ch.7
//     PlcTask Outputs/GVL_iXlinker.EtherCAT_Master_ATxxxx.Beckhoff_AT1xxx.Beckhoff_AT2xxxEK1122.A_0027_AT2020_0250_0021.CC_Outputs.Current_setpoint_value_Ch[7] <-> CC Outputs/Current setpoint value Ch.8
//     PlcTask Outputs/GVL_iXlinker.EtherCAT_Master_ATxxxx.Beckhoff_AT1xxx.Beckhoff_AT2xxxEK1122.A_0027_AT2020_0250_0021.CC_Outputs.Current_setpoint_value_Ch[8] <-> CC Outputs/Current setpoint value Ch.9
//     PlcTask Outputs/GVL_iXlinker.EtherCAT_Master_ATxxxx.Beckhoff_AT1xxx.Beckhoff_AT2xxxEK1122.A_0027_AT2020_0250_0021.CC_Outputs.Current_setpoint_value_Ch[9] <-> CC Outputs/Current setpoint value Ch.10
//     PlcTask Outputs/GVL_iXlinker.EtherCAT_Master_ATxxxx.Beckhoff_AT1xxx.Beckhoff_AT2xxxEK1122.A_0027_AT2020_0250_0021.CC_Outputs.Current_setpoint_value_Ch[10] <-> CC Outputs/Current setpoint value Ch.11
//     PlcTask Outputs/GVL_iXlinker.EtherCAT_Master_ATxxxx.Beckhoff_AT1xxx.Beckhoff_AT2xxxEK1122.A_0027_AT2020_0250_0021.CC_Outputs.Current_setpoint_value_Ch[11] <-> CC Outputs/Current setpoint value Ch.12
//     PlcTask Outputs/GVL_iXlinker.EtherCAT_Master_ATxxxx.Beckhoff_AT1xxx.Beckhoff_AT2xxxEK1122.A_0027_AT2020_0250_0021.CC_Outputs.Current_setpoint_value_Ch[12] <-> CC Outputs/Current setpoint value Ch.13
//     PlcTask Outputs/GVL_iXlinker.EtherCAT_Master_ATxxxx.Beckhoff_AT1xxx.Beckhoff_AT2xxxEK1122.A_0027_AT2020_0250_0021.CC_Outputs.Current_setpoint_value_Ch[13] <-> CC Outputs/Current setpoint value Ch.14
//     PlcTask Outputs/GVL_iXlinker.EtherCAT_Master_ATxxxx.Beckhoff_AT1xxx.Beckhoff_AT2xxxEK1122.A_0027_AT2020_0250_0021.CC_Outputs.Current_setpoint_value_Ch[14] <-> CC Outputs/Current setpoint value Ch.15
//     PlcTask Inputs/GVL_iXlinker.EtherCAT_Master_ATxxxx.Beckhoff_AT1xxx.Beckhoff_AT2xxxEK1122.A_0027_AT2020_0250_0021.WcState.WcState <-> WcState/WcState
//     PlcTask Inputs/GVL_iXlinker.EtherCAT_Master_ATxxxx.Beckhoff_AT1xxx.Beckhoff_AT2xxxEK1122.A_0027_AT2020_0250_0021.WcState.InputToggle <-> WcState/InputToggle
//     PlcTask Inputs/GVL_iXlinker.EtherCAT_Master_ATxxxx.Beckhoff_AT1xxx.Beckhoff_AT2xxxEK1122.A_0027_AT2020_0250_0021.InfoData.AdsAddr <-> InfoData/AdsAddr
//     PlcTask Inputs/GVL_iXlinker.EtherCAT_Master_ATxxxx.Beckhoff_AT1xxx.Beckhoff_AT2xxxEK1122.A_0027_AT2020_0250_0021.InfoData.DcOutputShift <-> InfoData/DcOutputShift
//     PlcTask Inputs/GVL_iXlinker.EtherCAT_Master_ATxxxx.Beckhoff_AT1xxx.Beckhoff_AT2xxxEK1122.A_0027_AT2020_0250_0021.InfoData.DcInputShift <-> InfoData/DcInputShift
//     PlcTask Inputs/GVL_iXlinker.EtherCAT_Master_ATxxxx.Beckhoff_AT1xxx.Beckhoff_AT2xxxEK1122.A_0027_AT2020_0250_0021.InfoData.State <-> InfoData/State
//   PLC/PLC Instance <-> EtherCAT Master ATxxxx/Beckhoff AT1xxx/Beckhoff AT2xxxEK1122/A_0028(AT2021-0250-0018)
//     PlcTask Inputs/GVL_iXlinker.EtherCAT_Master_ATxxxx.Beckhoff_AT1xxx.Beckhoff_AT2xxxEK1122.A_0028_AT2021_0250_0018.CC_Inputs.Status <-> CC Inputs/Status
//     PlcTask Inputs/GVL_iXlinker.EtherCAT_Master_ATxxxx.Beckhoff_AT1xxx.Beckhoff_AT2xxxEK1122.A_0028_AT2021_0250_0018.CC_Inputs.Current_actual_value_Ch[0] <-> CC Inputs/Current actual value Ch.1
//     PlcTask Inputs/GVL_iXlinker.EtherCAT_Master_ATxxxx.Beckhoff_AT1xxx.Beckhoff_AT2xxxEK1122.A_0028_AT2021_0250_0018.CC_Inputs.Current_actual_value_Ch[1] <-> CC Inputs/Current actual value Ch.2
//     PlcTask Inputs/GVL_iXlinker.EtherCAT_Master_ATxxxx.Beckhoff_AT1xxx.Beckhoff_AT2xxxEK1122.A_0028_AT2021_0250_0018.CC_Inputs.Current_actual_value_Ch[2] <-> CC Inputs/Current actual value Ch.3
//     PlcTask Inputs/GVL_iXlinker.EtherCAT_Master_ATxxxx.Beckhoff_AT1xxx.Beckhoff_AT2xxxEK1122.A_0028_AT2021_0250_0018.CC_Inputs.Current_actual_value_Ch[3] <-> CC Inputs/Current actual value Ch.4
//     PlcTask Inputs/GVL_iXlinker.EtherCAT_Master_ATxxxx.Beckhoff_AT1xxx.Beckhoff_AT2xxxEK1122.A_0028_AT2021_0250_0018.CC_Inputs.Current_actual_value_Ch[4] <-> CC Inputs/Current actual value Ch.5
//     PlcTask Inputs/GVL_iXlinker.EtherCAT_Master_ATxxxx.Beckhoff_AT1xxx.Beckhoff_AT2xxxEK1122.A_0028_AT2021_0250_0018.CC_Inputs.Current_actual_value_Ch[5] <-> CC Inputs/Current actual value Ch.6
//     PlcTask Inputs/GVL_iXlinker.EtherCAT_Master_ATxxxx.Beckhoff_AT1xxx.Beckhoff_AT2xxxEK1122.A_0028_AT2021_0250_0018.CC_Inputs.Current_actual_value_Ch[6] <-> CC Inputs/Current actual value Ch.7
//     PlcTask Inputs/GVL_iXlinker.EtherCAT_Master_ATxxxx.Beckhoff_AT1xxx.Beckhoff_AT2xxxEK1122.A_0028_AT2021_0250_0018.CC_Inputs.Current_actual_value_Ch[7] <-> CC Inputs/Current actual value Ch.8
//     PlcTask Inputs/GVL_iXlinker.EtherCAT_Master_ATxxxx.Beckhoff_AT1xxx.Beckhoff_AT2xxxEK1122.A_0028_AT2021_0250_0018.CC_Inputs.Current_actual_value_Ch[8] <-> CC Inputs/Current actual value Ch.9
//     PlcTask Inputs/GVL_iXlinker.EtherCAT_Master_ATxxxx.Beckhoff_AT1xxx.Beckhoff_AT2xxxEK1122.A_0028_AT2021_0250_0018.CC_Inputs.Current_actual_value_Ch[9] <-> CC Inputs/Current actual value Ch.10
//     PlcTask Inputs/GVL_iXlinker.EtherCAT_Master_ATxxxx.Beckhoff_AT1xxx.Beckhoff_AT2xxxEK1122.A_0028_AT2021_0250_0018.CC_Inputs.Current_actual_value_Ch[10] <-> CC Inputs/Current actual value Ch.11
//     PlcTask Inputs/GVL_iXlinker.EtherCAT_Master_ATxxxx.Beckhoff_AT1xxx.Beckhoff_AT2xxxEK1122.A_0028_AT2021_0250_0018.CC_Inputs.Current_actual_value_Ch[11] <-> CC Inputs/Current actual value Ch.12
//     PlcTask Inputs/GVL_iXlinker.EtherCAT_Master_ATxxxx.Beckhoff_AT1xxx.Beckhoff_AT2xxxEK1122.A_0028_AT2021_0250_0018.CC_Inputs.Current_actual_value_Ch[12] <-> CC Inputs/Current actual value Ch.13
//     PlcTask Inputs/GVL_iXlinker.EtherCAT_Master_ATxxxx.Beckhoff_AT1xxx.Beckhoff_AT2xxxEK1122.A_0028_AT2021_0250_0018.CC_Inputs.Current_actual_value_Ch[13] <-> CC Inputs/Current actual value Ch.14
//     PlcTask Inputs/GVL_iXlinker.EtherCAT_Master_ATxxxx.Beckhoff_AT1xxx.Beckhoff_AT2xxxEK1122.A_0028_AT2021_0250_0018.CC_Inputs.Current_actual_value_Ch[14] <-> CC Inputs/Current actual value Ch.15
//     PlcTask Outputs/GVL_iXlinker.EtherCAT_Master_ATxxxx.Beckhoff_AT1xxx.Beckhoff_AT2xxxEK1122.A_0028_AT2021_0250_0018.CC_Outputs.Control <-> CC Outputs/Control
//     PlcTask Outputs/GVL_iXlinker.EtherCAT_Master_ATxxxx.Beckhoff_AT1xxx.Beckhoff_AT2xxxEK1122.A_0028_AT2021_0250_0018.CC_Outputs.Current_setpoint_value_Ch[0] <-> CC Outputs/Current setpoint value Ch.1
//     PlcTask Outputs/GVL_iXlinker.EtherCAT_Master_ATxxxx.Beckhoff_AT1xxx.Beckhoff_AT2xxxEK1122.A_0028_AT2021_0250_0018.CC_Outputs.Current_setpoint_value_Ch[1] <-> CC Outputs/Current setpoint value Ch.2
//     PlcTask Outputs/GVL_iXlinker.EtherCAT_Master_ATxxxx.Beckhoff_AT1xxx.Beckhoff_AT2xxxEK1122.A_0028_AT2021_0250_0018.CC_Outputs.Current_setpoint_value_Ch[2] <-> CC Outputs/Current setpoint value Ch.3
//     PlcTask Outputs/GVL_iXlinker.EtherCAT_Master_ATxxxx.Beckhoff_AT1xxx.Beckhoff_AT2xxxEK1122.A_0028_AT2021_0250_0018.CC_Outputs.Current_setpoint_value_Ch[3] <-> CC Outputs/Current setpoint value Ch.4
//     PlcTask Outputs/GVL_iXlinker.EtherCAT_Master_ATxxxx.Beckhoff_AT1xxx.Beckhoff_AT2xxxEK1122.A_0028_AT2021_0250_0018.CC_Outputs.Current_setpoint_value_Ch[4] <-> CC Outputs/Current setpoint value Ch.5
//     PlcTask Outputs/GVL_iXlinker.EtherCAT_Master_ATxxxx.Beckhoff_AT1xxx.Beckhoff_AT2xxxEK1122.A_0028_AT2021_0250_0018.CC_Outputs.Current_setpoint_value_Ch[5] <-> CC Outputs/Current setpoint value Ch.6
//     PlcTask Outputs/GVL_iXlinker.EtherCAT_Master_ATxxxx.Beckhoff_AT1xxx.Beckhoff_AT2xxxEK1122.A_0028_AT2021_0250_0018.CC_Outputs.Current_setpoint_value_Ch[6] <-> CC Outputs/Current setpoint value Ch.7
//     PlcTask Outputs/GVL_iXlinker.EtherCAT_Master_ATxxxx.Beckhoff_AT1xxx.Beckhoff_AT2xxxEK1122.A_0028_AT2021_0250_0018.CC_Outputs.Current_setpoint_value_Ch[7] <-> CC Outputs/Current setpoint value Ch.8
//     PlcTask Outputs/GVL_iXlinker.EtherCAT_Master_ATxxxx.Beckhoff_AT1xxx.Beckhoff_AT2xxxEK1122.A_0028_AT2021_0250_0018.CC_Outputs.Current_setpoint_value_Ch[8] <-> CC Outputs/Current setpoint value Ch.9
//     PlcTask Outputs/GVL_iXlinker.EtherCAT_Master_ATxxxx.Beckhoff_AT1xxx.Beckhoff_AT2xxxEK1122.A_0028_AT2021_0250_0018.CC_Outputs.Current_setpoint_value_Ch[9] <-> CC Outputs/Current setpoint value Ch.10
//     PlcTask Outputs/GVL_iXlinker.EtherCAT_Master_ATxxxx.Beckhoff_AT1xxx.Beckhoff_AT2xxxEK1122.A_0028_AT2021_0250_0018.CC_Outputs.Current_setpoint_value_Ch[10] <-> CC Outputs/Current setpoint value Ch.11
//     PlcTask Outputs/GVL_iXlinker.EtherCAT_Master_ATxxxx.Beckhoff_AT1xxx.Beckhoff_AT2xxxEK1122.A_0028_AT2021_0250_0018.CC_Outputs.Current_setpoint_value_Ch[11] <-> CC Outputs/Current setpoint value Ch.12
//     PlcTask Outputs/GVL_iXlinker.EtherCAT_Master_ATxxxx.Beckhoff_AT1xxx.Beckhoff_AT2xxxEK1122.A_0028_AT2021_0250_0018.CC_Outputs.Current_setpoint_value_Ch[12] <-> CC Outputs/Current setpoint value Ch.13
//     PlcTask Outputs/GVL_iXlinker.EtherCAT_Master_ATxxxx.Beckhoff_AT1xxx.Beckhoff_AT2xxxEK1122.A_0028_AT2021_0250_0018.CC_Outputs.Current_setpoint_value_Ch[13] <-> CC Outputs/Current setpoint value Ch.14
//     PlcTask Outputs/GVL_iXlinker.EtherCAT_Master_ATxxxx.Beckhoff_AT1xxx.Beckhoff_AT2xxxEK1122.A_0028_AT2021_0250_0018.CC_Outputs.Current_setpoint_value_Ch[14] <-> CC Outputs/Current setpoint value Ch.15
//     PlcTask Inputs/GVL_iXlinker.EtherCAT_Master_ATxxxx.Beckhoff_AT1xxx.Beckhoff_AT2xxxEK1122.A_0028_AT2021_0250_0018.WcState.WcState <-> WcState/WcState
//     PlcTask Inputs/GVL_iXlinker.EtherCAT_Master_ATxxxx.Beckhoff_AT1xxx.Beckhoff_AT2xxxEK1122.A_0028_AT2021_0250_0018.WcState.InputToggle <-> WcState/InputToggle
//     PlcTask Inputs/GVL_iXlinker.EtherCAT_Master_ATxxxx.Beckhoff_AT1xxx.Beckhoff_AT2xxxEK1122.A_0028_AT2021_0250_0018.InfoData.AdsAddr <-> InfoData/AdsAddr
//     PlcTask Inputs/GVL_iXlinker.EtherCAT_Master_ATxxxx.Beckhoff_AT1xxx.Beckhoff_AT2xxxEK1122.A_0028_AT2021_0250_0018.InfoData.DcOutputShift <-> InfoData/DcOutputShift
//     PlcTask Inputs/GVL_iXlinker.EtherCAT_Master_ATxxxx.Beckhoff_AT1xxx.Beckhoff_AT2xxxEK1122.A_0028_AT2021_0250_0018.InfoData.DcInputShift <-> InfoData/DcInputShift
//     PlcTask Inputs/GVL_iXlinker.EtherCAT_Master_ATxxxx.Beckhoff_AT1xxx.Beckhoff_AT2xxxEK1122.A_0028_AT2021_0250_0018.InfoData.State <-> InfoData/State
//   PLC/PLC Instance <-> EtherCAT Master ATxxxx/Beckhoff AT1xxx/Beckhoff AT2xxxEK1122/A_0029(AT2021-0250-0020)
//     PlcTask Inputs/GVL_iXlinker.EtherCAT_Master_ATxxxx.Beckhoff_AT1xxx.Beckhoff_AT2xxxEK1122.A_0029_AT2021_0250_0020.CC_Inputs.Status <-> CC Inputs/Status
//     PlcTask Inputs/GVL_iXlinker.EtherCAT_Master_ATxxxx.Beckhoff_AT1xxx.Beckhoff_AT2xxxEK1122.A_0029_AT2021_0250_0020.CC_Inputs.Current_actual_value_Ch[0] <-> CC Inputs/Current actual value Ch.1
//     PlcTask Inputs/GVL_iXlinker.EtherCAT_Master_ATxxxx.Beckhoff_AT1xxx.Beckhoff_AT2xxxEK1122.A_0029_AT2021_0250_0020.CC_Inputs.Current_actual_value_Ch[1] <-> CC Inputs/Current actual value Ch.2
//     PlcTask Inputs/GVL_iXlinker.EtherCAT_Master_ATxxxx.Beckhoff_AT1xxx.Beckhoff_AT2xxxEK1122.A_0029_AT2021_0250_0020.CC_Inputs.Current_actual_value_Ch[2] <-> CC Inputs/Current actual value Ch.3
//     PlcTask Inputs/GVL_iXlinker.EtherCAT_Master_ATxxxx.Beckhoff_AT1xxx.Beckhoff_AT2xxxEK1122.A_0029_AT2021_0250_0020.CC_Inputs.Current_actual_value_Ch[3] <-> CC Inputs/Current actual value Ch.4
//     PlcTask Inputs/GVL_iXlinker.EtherCAT_Master_ATxxxx.Beckhoff_AT1xxx.Beckhoff_AT2xxxEK1122.A_0029_AT2021_0250_0020.CC_Inputs.Current_actual_value_Ch[4] <-> CC Inputs/Current actual value Ch.5
//     PlcTask Inputs/GVL_iXlinker.EtherCAT_Master_ATxxxx.Beckhoff_AT1xxx.Beckhoff_AT2xxxEK1122.A_0029_AT2021_0250_0020.CC_Inputs.Current_actual_value_Ch[5] <-> CC Inputs/Current actual value Ch.6
//     PlcTask Inputs/GVL_iXlinker.EtherCAT_Master_ATxxxx.Beckhoff_AT1xxx.Beckhoff_AT2xxxEK1122.A_0029_AT2021_0250_0020.CC_Inputs.Current_actual_value_Ch[6] <-> CC Inputs/Current actual value Ch.7
//     PlcTask Inputs/GVL_iXlinker.EtherCAT_Master_ATxxxx.Beckhoff_AT1xxx.Beckhoff_AT2xxxEK1122.A_0029_AT2021_0250_0020.CC_Inputs.Current_actual_value_Ch[7] <-> CC Inputs/Current actual value Ch.8
//     PlcTask Inputs/GVL_iXlinker.EtherCAT_Master_ATxxxx.Beckhoff_AT1xxx.Beckhoff_AT2xxxEK1122.A_0029_AT2021_0250_0020.CC_Inputs.Current_actual_value_Ch[8] <-> CC Inputs/Current actual value Ch.9
//     PlcTask Inputs/GVL_iXlinker.EtherCAT_Master_ATxxxx.Beckhoff_AT1xxx.Beckhoff_AT2xxxEK1122.A_0029_AT2021_0250_0020.CC_Inputs.Current_actual_value_Ch[9] <-> CC Inputs/Current actual value Ch.10
//     PlcTask Inputs/GVL_iXlinker.EtherCAT_Master_ATxxxx.Beckhoff_AT1xxx.Beckhoff_AT2xxxEK1122.A_0029_AT2021_0250_0020.CC_Inputs.Current_actual_value_Ch[10] <-> CC Inputs/Current actual value Ch.11
//     PlcTask Inputs/GVL_iXlinker.EtherCAT_Master_ATxxxx.Beckhoff_AT1xxx.Beckhoff_AT2xxxEK1122.A_0029_AT2021_0250_0020.CC_Inputs.Current_actual_value_Ch[11] <-> CC Inputs/Current actual value Ch.12
//     PlcTask Inputs/GVL_iXlinker.EtherCAT_Master_ATxxxx.Beckhoff_AT1xxx.Beckhoff_AT2xxxEK1122.A_0029_AT2021_0250_0020.CC_Inputs.Current_actual_value_Ch[12] <-> CC Inputs/Current actual value Ch.13
//     PlcTask Inputs/GVL_iXlinker.EtherCAT_Master_ATxxxx.Beckhoff_AT1xxx.Beckhoff_AT2xxxEK1122.A_0029_AT2021_0250_0020.CC_Inputs.Current_actual_value_Ch[13] <-> CC Inputs/Current actual value Ch.14
//     PlcTask Inputs/GVL_iXlinker.EtherCAT_Master_ATxxxx.Beckhoff_AT1xxx.Beckhoff_AT2xxxEK1122.A_0029_AT2021_0250_0020.CC_Inputs.Current_actual_value_Ch[14] <-> CC Inputs/Current actual value Ch.15
//     PlcTask Outputs/GVL_iXlinker.EtherCAT_Master_ATxxxx.Beckhoff_AT1xxx.Beckhoff_AT2xxxEK1122.A_0029_AT2021_0250_0020.CC_Outputs.Control <-> CC Outputs/Control
//     PlcTask Outputs/GVL_iXlinker.EtherCAT_Master_ATxxxx.Beckhoff_AT1xxx.Beckhoff_AT2xxxEK1122.A_0029_AT2021_0250_0020.CC_Outputs.Current_setpoint_value_Ch[0] <-> CC Outputs/Current setpoint value Ch.1
//     PlcTask Outputs/GVL_iXlinker.EtherCAT_Master_ATxxxx.Beckhoff_AT1xxx.Beckhoff_AT2xxxEK1122.A_0029_AT2021_0250_0020.CC_Outputs.Current_setpoint_value_Ch[1] <-> CC Outputs/Current setpoint value Ch.2
//     PlcTask Outputs/GVL_iXlinker.EtherCAT_Master_ATxxxx.Beckhoff_AT1xxx.Beckhoff_AT2xxxEK1122.A_0029_AT2021_0250_0020.CC_Outputs.Current_setpoint_value_Ch[2] <-> CC Outputs/Current setpoint value Ch.3
//     PlcTask Outputs/GVL_iXlinker.EtherCAT_Master_ATxxxx.Beckhoff_AT1xxx.Beckhoff_AT2xxxEK1122.A_0029_AT2021_0250_0020.CC_Outputs.Current_setpoint_value_Ch[3] <-> CC Outputs/Current setpoint value Ch.4
//     PlcTask Outputs/GVL_iXlinker.EtherCAT_Master_ATxxxx.Beckhoff_AT1xxx.Beckhoff_AT2xxxEK1122.A_0029_AT2021_0250_0020.CC_Outputs.Current_setpoint_value_Ch[4] <-> CC Outputs/Current setpoint value Ch.5
//     PlcTask Outputs/GVL_iXlinker.EtherCAT_Master_ATxxxx.Beckhoff_AT1xxx.Beckhoff_AT2xxxEK1122.A_0029_AT2021_0250_0020.CC_Outputs.Current_setpoint_value_Ch[5] <-> CC Outputs/Current setpoint value Ch.6
//     PlcTask Outputs/GVL_iXlinker.EtherCAT_Master_ATxxxx.Beckhoff_AT1xxx.Beckhoff_AT2xxxEK1122.A_0029_AT2021_0250_0020.CC_Outputs.Current_setpoint_value_Ch[6] <-> CC Outputs/Current setpoint value Ch.7
//     PlcTask Outputs/GVL_iXlinker.EtherCAT_Master_ATxxxx.Beckhoff_AT1xxx.Beckhoff_AT2xxxEK1122.A_0029_AT2021_0250_0020.CC_Outputs.Current_setpoint_value_Ch[7] <-> CC Outputs/Current setpoint value Ch.8
//     PlcTask Outputs/GVL_iXlinker.EtherCAT_Master_ATxxxx.Beckhoff_AT1xxx.Beckhoff_AT2xxxEK1122.A_0029_AT2021_0250_0020.CC_Outputs.Current_setpoint_value_Ch[8] <-> CC Outputs/Current setpoint value Ch.9
//     PlcTask Outputs/GVL_iXlinker.EtherCAT_Master_ATxxxx.Beckhoff_AT1xxx.Beckhoff_AT2xxxEK1122.A_0029_AT2021_0250_0020.CC_Outputs.Current_setpoint_value_Ch[9] <-> CC Outputs/Current setpoint value Ch.10
//     PlcTask Outputs/GVL_iXlinker.EtherCAT_Master_ATxxxx.Beckhoff_AT1xxx.Beckhoff_AT2xxxEK1122.A_0029_AT2021_0250_0020.CC_Outputs.Current_setpoint_value_Ch[10] <-> CC Outputs/Current setpoint value Ch.11
//     PlcTask Outputs/GVL_iXlinker.EtherCAT_Master_ATxxxx.Beckhoff_AT1xxx.Beckhoff_AT2xxxEK1122.A_0029_AT2021_0250_0020.CC_Outputs.Current_setpoint_value_Ch[11] <-> CC Outputs/Current setpoint value Ch.12
//     PlcTask Outputs/GVL_iXlinker.EtherCAT_Master_ATxxxx.Beckhoff_AT1xxx.Beckhoff_AT2xxxEK1122.A_0029_AT2021_0250_0020.CC_Outputs.Current_setpoint_value_Ch[12] <-> CC Outputs/Current setpoint value Ch.13
//     PlcTask Outputs/GVL_iXlinker.EtherCAT_Master_ATxxxx.Beckhoff_AT1xxx.Beckhoff_AT2xxxEK1122.A_0029_AT2021_0250_0020.CC_Outputs.Current_setpoint_value_Ch[13] <-> CC Outputs/Current setpoint value Ch.14
//     PlcTask Outputs/GVL_iXlinker.EtherCAT_Master_ATxxxx.Beckhoff_AT1xxx.Beckhoff_AT2xxxEK1122.A_0029_AT2021_0250_0020.CC_Outputs.Current_setpoint_value_Ch[14] <-> CC Outputs/Current setpoint value Ch.15
//     PlcTask Inputs/GVL_iXlinker.EtherCAT_Master_ATxxxx.Beckhoff_AT1xxx.Beckhoff_AT2xxxEK1122.A_0029_AT2021_0250_0020.WcState.WcState <-> WcState/WcState
//     PlcTask Inputs/GVL_iXlinker.EtherCAT_Master_ATxxxx.Beckhoff_AT1xxx.Beckhoff_AT2xxxEK1122.A_0029_AT2021_0250_0020.WcState.InputToggle <-> WcState/InputToggle
//     PlcTask Inputs/GVL_iXlinker.EtherCAT_Master_ATxxxx.Beckhoff_AT1xxx.Beckhoff_AT2xxxEK1122.A_0029_AT2021_0250_0020.InfoData.AdsAddr <-> InfoData/AdsAddr
//     PlcTask Inputs/GVL_iXlinker.EtherCAT_Master_ATxxxx.Beckhoff_AT1xxx.Beckhoff_AT2xxxEK1122.A_0029_AT2021_0250_0020.InfoData.DcOutputShift <-> InfoData/DcOutputShift
//     PlcTask Inputs/GVL_iXlinker.EtherCAT_Master_ATxxxx.Beckhoff_AT1xxx.Beckhoff_AT2xxxEK1122.A_0029_AT2021_0250_0020.InfoData.DcInputShift <-> InfoData/DcInputShift
//     PlcTask Inputs/GVL_iXlinker.EtherCAT_Master_ATxxxx.Beckhoff_AT1xxx.Beckhoff_AT2xxxEK1122.A_0029_AT2021_0250_0020.InfoData.State <-> InfoData/State
//   PLC/PLC Instance <-> EtherCAT Master ATxxxx/Beckhoff AT1xxx/Beckhoff AT2xxxEK1122/A_0030(AT2025-0250-0018)
//     PlcTask Inputs/GVL_iXlinker.EtherCAT_Master_ATxxxx.Beckhoff_AT1xxx.Beckhoff_AT2xxxEK1122.A_0030_AT2025_0250_0018.CC_Inputs.Status <-> CC Inputs/Status
//     PlcTask Inputs/GVL_iXlinker.EtherCAT_Master_ATxxxx.Beckhoff_AT1xxx.Beckhoff_AT2xxxEK1122.A_0030_AT2025_0250_0018.CC_Inputs.Current_actual_value_Ch[0] <-> CC Inputs/Current actual value Ch.1
//     PlcTask Inputs/GVL_iXlinker.EtherCAT_Master_ATxxxx.Beckhoff_AT1xxx.Beckhoff_AT2xxxEK1122.A_0030_AT2025_0250_0018.CC_Inputs.Current_actual_value_Ch[1] <-> CC Inputs/Current actual value Ch.2
//     PlcTask Inputs/GVL_iXlinker.EtherCAT_Master_ATxxxx.Beckhoff_AT1xxx.Beckhoff_AT2xxxEK1122.A_0030_AT2025_0250_0018.CC_Inputs.Current_actual_value_Ch[2] <-> CC Inputs/Current actual value Ch.3
//     PlcTask Inputs/GVL_iXlinker.EtherCAT_Master_ATxxxx.Beckhoff_AT1xxx.Beckhoff_AT2xxxEK1122.A_0030_AT2025_0250_0018.CC_Inputs.Current_actual_value_Ch[3] <-> CC Inputs/Current actual value Ch.4
//     PlcTask Inputs/GVL_iXlinker.EtherCAT_Master_ATxxxx.Beckhoff_AT1xxx.Beckhoff_AT2xxxEK1122.A_0030_AT2025_0250_0018.CC_Inputs.Current_actual_value_Ch[4] <-> CC Inputs/Current actual value Ch.5
//     PlcTask Inputs/GVL_iXlinker.EtherCAT_Master_ATxxxx.Beckhoff_AT1xxx.Beckhoff_AT2xxxEK1122.A_0030_AT2025_0250_0018.CC_Inputs.Current_actual_value_Ch[5] <-> CC Inputs/Current actual value Ch.6
//     PlcTask Inputs/GVL_iXlinker.EtherCAT_Master_ATxxxx.Beckhoff_AT1xxx.Beckhoff_AT2xxxEK1122.A_0030_AT2025_0250_0018.CC_Inputs.Current_actual_value_Ch[6] <-> CC Inputs/Current actual value Ch.7
//     PlcTask Inputs/GVL_iXlinker.EtherCAT_Master_ATxxxx.Beckhoff_AT1xxx.Beckhoff_AT2xxxEK1122.A_0030_AT2025_0250_0018.CC_Inputs.Current_actual_value_Ch[7] <-> CC Inputs/Current actual value Ch.8
//     PlcTask Inputs/GVL_iXlinker.EtherCAT_Master_ATxxxx.Beckhoff_AT1xxx.Beckhoff_AT2xxxEK1122.A_0030_AT2025_0250_0018.CC_Inputs.Current_actual_value_Ch[8] <-> CC Inputs/Current actual value Ch.9
//     PlcTask Inputs/GVL_iXlinker.EtherCAT_Master_ATxxxx.Beckhoff_AT1xxx.Beckhoff_AT2xxxEK1122.A_0030_AT2025_0250_0018.CC_Inputs.Current_actual_value_Ch[9] <-> CC Inputs/Current actual value Ch.10
//     PlcTask Inputs/GVL_iXlinker.EtherCAT_Master_ATxxxx.Beckhoff_AT1xxx.Beckhoff_AT2xxxEK1122.A_0030_AT2025_0250_0018.CC_Inputs.Current_actual_value_Ch[10] <-> CC Inputs/Current actual value Ch.11
//     PlcTask Inputs/GVL_iXlinker.EtherCAT_Master_ATxxxx.Beckhoff_AT1xxx.Beckhoff_AT2xxxEK1122.A_0030_AT2025_0250_0018.CC_Inputs.Current_actual_value_Ch[11] <-> CC Inputs/Current actual value Ch.12
//     PlcTask Inputs/GVL_iXlinker.EtherCAT_Master_ATxxxx.Beckhoff_AT1xxx.Beckhoff_AT2xxxEK1122.A_0030_AT2025_0250_0018.CC_Inputs.Current_actual_value_Ch[12] <-> CC Inputs/Current actual value Ch.13
//     PlcTask Inputs/GVL_iXlinker.EtherCAT_Master_ATxxxx.Beckhoff_AT1xxx.Beckhoff_AT2xxxEK1122.A_0030_AT2025_0250_0018.CC_Inputs.Current_actual_value_Ch[13] <-> CC Inputs/Current actual value Ch.14
//     PlcTask Inputs/GVL_iXlinker.EtherCAT_Master_ATxxxx.Beckhoff_AT1xxx.Beckhoff_AT2xxxEK1122.A_0030_AT2025_0250_0018.CC_Inputs.Current_actual_value_Ch[14] <-> CC Inputs/Current actual value Ch.15
//     PlcTask Outputs/GVL_iXlinker.EtherCAT_Master_ATxxxx.Beckhoff_AT1xxx.Beckhoff_AT2xxxEK1122.A_0030_AT2025_0250_0018.CC_Outputs.Control <-> CC Outputs/Control
//     PlcTask Outputs/GVL_iXlinker.EtherCAT_Master_ATxxxx.Beckhoff_AT1xxx.Beckhoff_AT2xxxEK1122.A_0030_AT2025_0250_0018.CC_Outputs.Current_setpoint_value_Ch[0] <-> CC Outputs/Current setpoint value Ch.1
//     PlcTask Outputs/GVL_iXlinker.EtherCAT_Master_ATxxxx.Beckhoff_AT1xxx.Beckhoff_AT2xxxEK1122.A_0030_AT2025_0250_0018.CC_Outputs.Current_setpoint_value_Ch[1] <-> CC Outputs/Current setpoint value Ch.2
//     PlcTask Outputs/GVL_iXlinker.EtherCAT_Master_ATxxxx.Beckhoff_AT1xxx.Beckhoff_AT2xxxEK1122.A_0030_AT2025_0250_0018.CC_Outputs.Current_setpoint_value_Ch[2] <-> CC Outputs/Current setpoint value Ch.3
//     PlcTask Outputs/GVL_iXlinker.EtherCAT_Master_ATxxxx.Beckhoff_AT1xxx.Beckhoff_AT2xxxEK1122.A_0030_AT2025_0250_0018.CC_Outputs.Current_setpoint_value_Ch[3] <-> CC Outputs/Current setpoint value Ch.4
//     PlcTask Outputs/GVL_iXlinker.EtherCAT_Master_ATxxxx.Beckhoff_AT1xxx.Beckhoff_AT2xxxEK1122.A_0030_AT2025_0250_0018.CC_Outputs.Current_setpoint_value_Ch[4] <-> CC Outputs/Current setpoint value Ch.5
//     PlcTask Outputs/GVL_iXlinker.EtherCAT_Master_ATxxxx.Beckhoff_AT1xxx.Beckhoff_AT2xxxEK1122.A_0030_AT2025_0250_0018.CC_Outputs.Current_setpoint_value_Ch[5] <-> CC Outputs/Current setpoint value Ch.6
//     PlcTask Outputs/GVL_iXlinker.EtherCAT_Master_ATxxxx.Beckhoff_AT1xxx.Beckhoff_AT2xxxEK1122.A_0030_AT2025_0250_0018.CC_Outputs.Current_setpoint_value_Ch[6] <-> CC Outputs/Current setpoint value Ch.7
//     PlcTask Outputs/GVL_iXlinker.EtherCAT_Master_ATxxxx.Beckhoff_AT1xxx.Beckhoff_AT2xxxEK1122.A_0030_AT2025_0250_0018.CC_Outputs.Current_setpoint_value_Ch[7] <-> CC Outputs/Current setpoint value Ch.8
//     PlcTask Outputs/GVL_iXlinker.EtherCAT_Master_ATxxxx.Beckhoff_AT1xxx.Beckhoff_AT2xxxEK1122.A_0030_AT2025_0250_0018.CC_Outputs.Current_setpoint_value_Ch[8] <-> CC Outputs/Current setpoint value Ch.9
//     PlcTask Outputs/GVL_iXlinker.EtherCAT_Master_ATxxxx.Beckhoff_AT1xxx.Beckhoff_AT2xxxEK1122.A_0030_AT2025_0250_0018.CC_Outputs.Current_setpoint_value_Ch[9] <-> CC Outputs/Current setpoint value Ch.10
//     PlcTask Outputs/GVL_iXlinker.EtherCAT_Master_ATxxxx.Beckhoff_AT1xxx.Beckhoff_AT2xxxEK1122.A_0030_AT2025_0250_0018.CC_Outputs.Current_setpoint_value_Ch[10] <-> CC Outputs/Current setpoint value Ch.11
//     PlcTask Outputs/GVL_iXlinker.EtherCAT_Master_ATxxxx.Beckhoff_AT1xxx.Beckhoff_AT2xxxEK1122.A_0030_AT2025_0250_0018.CC_Outputs.Current_setpoint_value_Ch[11] <-> CC Outputs/Current setpoint value Ch.12
//     PlcTask Outputs/GVL_iXlinker.EtherCAT_Master_ATxxxx.Beckhoff_AT1xxx.Beckhoff_AT2xxxEK1122.A_0030_AT2025_0250_0018.CC_Outputs.Current_setpoint_value_Ch[12] <-> CC Outputs/Current setpoint value Ch.13
//     PlcTask Outputs/GVL_iXlinker.EtherCAT_Master_ATxxxx.Beckhoff_AT1xxx.Beckhoff_AT2xxxEK1122.A_0030_AT2025_0250_0018.CC_Outputs.Current_setpoint_value_Ch[13] <-> CC Outputs/Current setpoint value Ch.14
//     PlcTask Outputs/GVL_iXlinker.EtherCAT_Master_ATxxxx.Beckhoff_AT1xxx.Beckhoff_AT2xxxEK1122.A_0030_AT2025_0250_0018.CC_Outputs.Current_setpoint_value_Ch[14] <-> CC Outputs/Current setpoint value Ch.15
//     PlcTask Inputs/GVL_iXlinker.EtherCAT_Master_ATxxxx.Beckhoff_AT1xxx.Beckhoff_AT2xxxEK1122.A_0030_AT2025_0250_0018.WcState.WcState <-> WcState/WcState
//     PlcTask Inputs/GVL_iXlinker.EtherCAT_Master_ATxxxx.Beckhoff_AT1xxx.Beckhoff_AT2xxxEK1122.A_0030_AT2025_0250_0018.WcState.InputToggle <-> WcState/InputToggle
//     PlcTask Inputs/GVL_iXlinker.EtherCAT_Master_ATxxxx.Beckhoff_AT1xxx.Beckhoff_AT2xxxEK1122.A_0030_AT2025_0250_0018.InfoData.AdsAddr <-> InfoData/AdsAddr
//     PlcTask Inputs/GVL_iXlinker.EtherCAT_Master_ATxxxx.Beckhoff_AT1xxx.Beckhoff_AT2xxxEK1122.A_0030_AT2025_0250_0018.InfoData.DcOutputShift <-> InfoData/DcOutputShift
//     PlcTask Inputs/GVL_iXlinker.EtherCAT_Master_ATxxxx.Beckhoff_AT1xxx.Beckhoff_AT2xxxEK1122.A_0030_AT2025_0250_0018.InfoData.DcInputShift <-> InfoData/DcInputShift
//     PlcTask Inputs/GVL_iXlinker.EtherCAT_Master_ATxxxx.Beckhoff_AT1xxx.Beckhoff_AT2xxxEK1122.A_0030_AT2025_0250_0018.InfoData.State <-> InfoData/State
//   PLC/PLC Instance <-> EtherCAT Master ATxxxx/Beckhoff AT1xxx/Beckhoff AT2xxxEK1122/A_0031(AT2026-0250-0021)
//     PlcTask Inputs/GVL_iXlinker.EtherCAT_Master_ATxxxx.Beckhoff_AT1xxx.Beckhoff_AT2xxxEK1122.A_0031_AT2026_0250_0021.CC_Inputs.Status <-> CC Inputs/Status
//     PlcTask Inputs/GVL_iXlinker.EtherCAT_Master_ATxxxx.Beckhoff_AT1xxx.Beckhoff_AT2xxxEK1122.A_0031_AT2026_0250_0021.CC_Inputs.Current_actual_value_Ch[0] <-> CC Inputs/Current actual value Ch.1
//     PlcTask Inputs/GVL_iXlinker.EtherCAT_Master_ATxxxx.Beckhoff_AT1xxx.Beckhoff_AT2xxxEK1122.A_0031_AT2026_0250_0021.CC_Inputs.Current_actual_value_Ch[1] <-> CC Inputs/Current actual value Ch.2
//     PlcTask Inputs/GVL_iXlinker.EtherCAT_Master_ATxxxx.Beckhoff_AT1xxx.Beckhoff_AT2xxxEK1122.A_0031_AT2026_0250_0021.CC_Inputs.Current_actual_value_Ch[2] <-> CC Inputs/Current actual value Ch.3
//     PlcTask Inputs/GVL_iXlinker.EtherCAT_Master_ATxxxx.Beckhoff_AT1xxx.Beckhoff_AT2xxxEK1122.A_0031_AT2026_0250_0021.CC_Inputs.Current_actual_value_Ch[3] <-> CC Inputs/Current actual value Ch.4
//     PlcTask Inputs/GVL_iXlinker.EtherCAT_Master_ATxxxx.Beckhoff_AT1xxx.Beckhoff_AT2xxxEK1122.A_0031_AT2026_0250_0021.CC_Inputs.Current_actual_value_Ch[4] <-> CC Inputs/Current actual value Ch.5
//     PlcTask Inputs/GVL_iXlinker.EtherCAT_Master_ATxxxx.Beckhoff_AT1xxx.Beckhoff_AT2xxxEK1122.A_0031_AT2026_0250_0021.CC_Inputs.Current_actual_value_Ch[5] <-> CC Inputs/Current actual value Ch.6
//     PlcTask Inputs/GVL_iXlinker.EtherCAT_Master_ATxxxx.Beckhoff_AT1xxx.Beckhoff_AT2xxxEK1122.A_0031_AT2026_0250_0021.CC_Inputs.Current_actual_value_Ch[6] <-> CC Inputs/Current actual value Ch.7
//     PlcTask Inputs/GVL_iXlinker.EtherCAT_Master_ATxxxx.Beckhoff_AT1xxx.Beckhoff_AT2xxxEK1122.A_0031_AT2026_0250_0021.CC_Inputs.Current_actual_value_Ch[7] <-> CC Inputs/Current actual value Ch.8
//     PlcTask Inputs/GVL_iXlinker.EtherCAT_Master_ATxxxx.Beckhoff_AT1xxx.Beckhoff_AT2xxxEK1122.A_0031_AT2026_0250_0021.CC_Inputs.Current_actual_value_Ch[8] <-> CC Inputs/Current actual value Ch.9
//     PlcTask Inputs/GVL_iXlinker.EtherCAT_Master_ATxxxx.Beckhoff_AT1xxx.Beckhoff_AT2xxxEK1122.A_0031_AT2026_0250_0021.CC_Inputs.Current_actual_value_Ch[9] <-> CC Inputs/Current actual value Ch.10
//     PlcTask Inputs/GVL_iXlinker.EtherCAT_Master_ATxxxx.Beckhoff_AT1xxx.Beckhoff_AT2xxxEK1122.A_0031_AT2026_0250_0021.CC_Inputs.Current_actual_value_Ch[10] <-> CC Inputs/Current actual value Ch.11
//     PlcTask Inputs/GVL_iXlinker.EtherCAT_Master_ATxxxx.Beckhoff_AT1xxx.Beckhoff_AT2xxxEK1122.A_0031_AT2026_0250_0021.CC_Inputs.Current_actual_value_Ch[11] <-> CC Inputs/Current actual value Ch.12
//     PlcTask Inputs/GVL_iXlinker.EtherCAT_Master_ATxxxx.Beckhoff_AT1xxx.Beckhoff_AT2xxxEK1122.A_0031_AT2026_0250_0021.CC_Inputs.Current_actual_value_Ch[12] <-> CC Inputs/Current actual value Ch.13
//     PlcTask Inputs/GVL_iXlinker.EtherCAT_Master_ATxxxx.Beckhoff_AT1xxx.Beckhoff_AT2xxxEK1122.A_0031_AT2026_0250_0021.CC_Inputs.Current_actual_value_Ch[13] <-> CC Inputs/Current actual value Ch.14
//     PlcTask Inputs/GVL_iXlinker.EtherCAT_Master_ATxxxx.Beckhoff_AT1xxx.Beckhoff_AT2xxxEK1122.A_0031_AT2026_0250_0021.CC_Inputs.Current_actual_value_Ch[14] <-> CC Inputs/Current actual value Ch.15
//     PlcTask Outputs/GVL_iXlinker.EtherCAT_Master_ATxxxx.Beckhoff_AT1xxx.Beckhoff_AT2xxxEK1122.A_0031_AT2026_0250_0021.CC_Outputs.Control <-> CC Outputs/Control
//     PlcTask Outputs/GVL_iXlinker.EtherCAT_Master_ATxxxx.Beckhoff_AT1xxx.Beckhoff_AT2xxxEK1122.A_0031_AT2026_0250_0021.CC_Outputs.Current_setpoint_value_Ch[0] <-> CC Outputs/Current setpoint value Ch.1
//     PlcTask Outputs/GVL_iXlinker.EtherCAT_Master_ATxxxx.Beckhoff_AT1xxx.Beckhoff_AT2xxxEK1122.A_0031_AT2026_0250_0021.CC_Outputs.Current_setpoint_value_Ch[1] <-> CC Outputs/Current setpoint value Ch.2
//     PlcTask Outputs/GVL_iXlinker.EtherCAT_Master_ATxxxx.Beckhoff_AT1xxx.Beckhoff_AT2xxxEK1122.A_0031_AT2026_0250_0021.CC_Outputs.Current_setpoint_value_Ch[2] <-> CC Outputs/Current setpoint value Ch.3
//     PlcTask Outputs/GVL_iXlinker.EtherCAT_Master_ATxxxx.Beckhoff_AT1xxx.Beckhoff_AT2xxxEK1122.A_0031_AT2026_0250_0021.CC_Outputs.Current_setpoint_value_Ch[3] <-> CC Outputs/Current setpoint value Ch.4
//     PlcTask Outputs/GVL_iXlinker.EtherCAT_Master_ATxxxx.Beckhoff_AT1xxx.Beckhoff_AT2xxxEK1122.A_0031_AT2026_0250_0021.CC_Outputs.Current_setpoint_value_Ch[4] <-> CC Outputs/Current setpoint value Ch.5
//     PlcTask Outputs/GVL_iXlinker.EtherCAT_Master_ATxxxx.Beckhoff_AT1xxx.Beckhoff_AT2xxxEK1122.A_0031_AT2026_0250_0021.CC_Outputs.Current_setpoint_value_Ch[5] <-> CC Outputs/Current setpoint value Ch.6
//     PlcTask Outputs/GVL_iXlinker.EtherCAT_Master_ATxxxx.Beckhoff_AT1xxx.Beckhoff_AT2xxxEK1122.A_0031_AT2026_0250_0021.CC_Outputs.Current_setpoint_value_Ch[6] <-> CC Outputs/Current setpoint value Ch.7
//     PlcTask Outputs/GVL_iXlinker.EtherCAT_Master_ATxxxx.Beckhoff_AT1xxx.Beckhoff_AT2xxxEK1122.A_0031_AT2026_0250_0021.CC_Outputs.Current_setpoint_value_Ch[7] <-> CC Outputs/Current setpoint value Ch.8
//     PlcTask Outputs/GVL_iXlinker.EtherCAT_Master_ATxxxx.Beckhoff_AT1xxx.Beckhoff_AT2xxxEK1122.A_0031_AT2026_0250_0021.CC_Outputs.Current_setpoint_value_Ch[8] <-> CC Outputs/Current setpoint value Ch.9
//     PlcTask Outputs/GVL_iXlinker.EtherCAT_Master_ATxxxx.Beckhoff_AT1xxx.Beckhoff_AT2xxxEK1122.A_0031_AT2026_0250_0021.CC_Outputs.Current_setpoint_value_Ch[9] <-> CC Outputs/Current setpoint value Ch.10
//     PlcTask Outputs/GVL_iXlinker.EtherCAT_Master_ATxxxx.Beckhoff_AT1xxx.Beckhoff_AT2xxxEK1122.A_0031_AT2026_0250_0021.CC_Outputs.Current_setpoint_value_Ch[10] <-> CC Outputs/Current setpoint value Ch.11
//     PlcTask Outputs/GVL_iXlinker.EtherCAT_Master_ATxxxx.Beckhoff_AT1xxx.Beckhoff_AT2xxxEK1122.A_0031_AT2026_0250_0021.CC_Outputs.Current_setpoint_value_Ch[11] <-> CC Outputs/Current setpoint value Ch.12
//     PlcTask Outputs/GVL_iXlinker.EtherCAT_Master_ATxxxx.Beckhoff_AT1xxx.Beckhoff_AT2xxxEK1122.A_0031_AT2026_0250_0021.CC_Outputs.Current_setpoint_value_Ch[12] <-> CC Outputs/Current setpoint value Ch.13
//     PlcTask Outputs/GVL_iXlinker.EtherCAT_Master_ATxxxx.Beckhoff_AT1xxx.Beckhoff_AT2xxxEK1122.A_0031_AT2026_0250_0021.CC_Outputs.Current_setpoint_value_Ch[13] <-> CC Outputs/Current setpoint value Ch.14
//     PlcTask Outputs/GVL_iXlinker.EtherCAT_Master_ATxxxx.Beckhoff_AT1xxx.Beckhoff_AT2xxxEK1122.A_0031_AT2026_0250_0021.CC_Outputs.Current_setpoint_value_Ch[14] <-> CC Outputs/Current setpoint value Ch.15
//     PlcTask Inputs/GVL_iXlinker.EtherCAT_Master_ATxxxx.Beckhoff_AT1xxx.Beckhoff_AT2xxxEK1122.A_0031_AT2026_0250_0021.WcState.WcState <-> WcState/WcState
//     PlcTask Inputs/GVL_iXlinker.EtherCAT_Master_ATxxxx.Beckhoff_AT1xxx.Beckhoff_AT2xxxEK1122.A_0031_AT2026_0250_0021.WcState.InputToggle <-> WcState/InputToggle
//     PlcTask Inputs/GVL_iXlinker.EtherCAT_Master_ATxxxx.Beckhoff_AT1xxx.Beckhoff_AT2xxxEK1122.A_0031_AT2026_0250_0021.InfoData.AdsAddr <-> InfoData/AdsAddr
//     PlcTask Inputs/GVL_iXlinker.EtherCAT_Master_ATxxxx.Beckhoff_AT1xxx.Beckhoff_AT2xxxEK1122.A_0031_AT2026_0250_0021.InfoData.DcOutputShift <-> InfoData/DcOutputShift
//     PlcTask Inputs/GVL_iXlinker.EtherCAT_Master_ATxxxx.Beckhoff_AT1xxx.Beckhoff_AT2xxxEK1122.A_0031_AT2026_0250_0021.InfoData.DcInputShift <-> InfoData/DcInputShift
//     PlcTask Inputs/GVL_iXlinker.EtherCAT_Master_ATxxxx.Beckhoff_AT1xxx.Beckhoff_AT2xxxEK1122.A_0031_AT2026_0250_0021.InfoData.State <-> InfoData/State
//   PLC/PLC Instance <-> EtherCAT Master ATxxxx/Beckhoff AT1xxx/Beckhoff AT2xxxEK1122/A_0032(AT2026-0250-0023)
//     PlcTask Inputs/GVL_iXlinker.EtherCAT_Master_ATxxxx.Beckhoff_AT1xxx.Beckhoff_AT2xxxEK1122.A_0032_AT2026_0250_0023.CC_Inputs.Status <-> CC Inputs/Status
//     PlcTask Inputs/GVL_iXlinker.EtherCAT_Master_ATxxxx.Beckhoff_AT1xxx.Beckhoff_AT2xxxEK1122.A_0032_AT2026_0250_0023.CC_Inputs.Current_actual_value_Ch[0] <-> CC Inputs/Current actual value Ch.1
//     PlcTask Inputs/GVL_iXlinker.EtherCAT_Master_ATxxxx.Beckhoff_AT1xxx.Beckhoff_AT2xxxEK1122.A_0032_AT2026_0250_0023.CC_Inputs.Current_actual_value_Ch[1] <-> CC Inputs/Current actual value Ch.2
//     PlcTask Inputs/GVL_iXlinker.EtherCAT_Master_ATxxxx.Beckhoff_AT1xxx.Beckhoff_AT2xxxEK1122.A_0032_AT2026_0250_0023.CC_Inputs.Current_actual_value_Ch[2] <-> CC Inputs/Current actual value Ch.3
//     PlcTask Inputs/GVL_iXlinker.EtherCAT_Master_ATxxxx.Beckhoff_AT1xxx.Beckhoff_AT2xxxEK1122.A_0032_AT2026_0250_0023.CC_Inputs.Current_actual_value_Ch[3] <-> CC Inputs/Current actual value Ch.4
//     PlcTask Inputs/GVL_iXlinker.EtherCAT_Master_ATxxxx.Beckhoff_AT1xxx.Beckhoff_AT2xxxEK1122.A_0032_AT2026_0250_0023.CC_Inputs.Current_actual_value_Ch[4] <-> CC Inputs/Current actual value Ch.5
//     PlcTask Inputs/GVL_iXlinker.EtherCAT_Master_ATxxxx.Beckhoff_AT1xxx.Beckhoff_AT2xxxEK1122.A_0032_AT2026_0250_0023.CC_Inputs.Current_actual_value_Ch[5] <-> CC Inputs/Current actual value Ch.6
//     PlcTask Inputs/GVL_iXlinker.EtherCAT_Master_ATxxxx.Beckhoff_AT1xxx.Beckhoff_AT2xxxEK1122.A_0032_AT2026_0250_0023.CC_Inputs.Current_actual_value_Ch[6] <-> CC Inputs/Current actual value Ch.7
//     PlcTask Inputs/GVL_iXlinker.EtherCAT_Master_ATxxxx.Beckhoff_AT1xxx.Beckhoff_AT2xxxEK1122.A_0032_AT2026_0250_0023.CC_Inputs.Current_actual_value_Ch[7] <-> CC Inputs/Current actual value Ch.8
//     PlcTask Inputs/GVL_iXlinker.EtherCAT_Master_ATxxxx.Beckhoff_AT1xxx.Beckhoff_AT2xxxEK1122.A_0032_AT2026_0250_0023.CC_Inputs.Current_actual_value_Ch[8] <-> CC Inputs/Current actual value Ch.9
//     PlcTask Inputs/GVL_iXlinker.EtherCAT_Master_ATxxxx.Beckhoff_AT1xxx.Beckhoff_AT2xxxEK1122.A_0032_AT2026_0250_0023.CC_Inputs.Current_actual_value_Ch[9] <-> CC Inputs/Current actual value Ch.10
//     PlcTask Inputs/GVL_iXlinker.EtherCAT_Master_ATxxxx.Beckhoff_AT1xxx.Beckhoff_AT2xxxEK1122.A_0032_AT2026_0250_0023.CC_Inputs.Current_actual_value_Ch[10] <-> CC Inputs/Current actual value Ch.11
//     PlcTask Inputs/GVL_iXlinker.EtherCAT_Master_ATxxxx.Beckhoff_AT1xxx.Beckhoff_AT2xxxEK1122.A_0032_AT2026_0250_0023.CC_Inputs.Current_actual_value_Ch[11] <-> CC Inputs/Current actual value Ch.12
//     PlcTask Inputs/GVL_iXlinker.EtherCAT_Master_ATxxxx.Beckhoff_AT1xxx.Beckhoff_AT2xxxEK1122.A_0032_AT2026_0250_0023.CC_Inputs.Current_actual_value_Ch[12] <-> CC Inputs/Current actual value Ch.13
//     PlcTask Inputs/GVL_iXlinker.EtherCAT_Master_ATxxxx.Beckhoff_AT1xxx.Beckhoff_AT2xxxEK1122.A_0032_AT2026_0250_0023.CC_Inputs.Current_actual_value_Ch[13] <-> CC Inputs/Current actual value Ch.14
//     PlcTask Inputs/GVL_iXlinker.EtherCAT_Master_ATxxxx.Beckhoff_AT1xxx.Beckhoff_AT2xxxEK1122.A_0032_AT2026_0250_0023.CC_Inputs.Current_actual_value_Ch[14] <-> CC Inputs/Current actual value Ch.15
//     PlcTask Outputs/GVL_iXlinker.EtherCAT_Master_ATxxxx.Beckhoff_AT1xxx.Beckhoff_AT2xxxEK1122.A_0032_AT2026_0250_0023.CC_Outputs.Control <-> CC Outputs/Control
//     PlcTask Outputs/GVL_iXlinker.EtherCAT_Master_ATxxxx.Beckhoff_AT1xxx.Beckhoff_AT2xxxEK1122.A_0032_AT2026_0250_0023.CC_Outputs.Current_setpoint_value_Ch[0] <-> CC Outputs/Current setpoint value Ch.1
//     PlcTask Outputs/GVL_iXlinker.EtherCAT_Master_ATxxxx.Beckhoff_AT1xxx.Beckhoff_AT2xxxEK1122.A_0032_AT2026_0250_0023.CC_Outputs.Current_setpoint_value_Ch[1] <-> CC Outputs/Current setpoint value Ch.2
//     PlcTask Outputs/GVL_iXlinker.EtherCAT_Master_ATxxxx.Beckhoff_AT1xxx.Beckhoff_AT2xxxEK1122.A_0032_AT2026_0250_0023.CC_Outputs.Current_setpoint_value_Ch[2] <-> CC Outputs/Current setpoint value Ch.3
//     PlcTask Outputs/GVL_iXlinker.EtherCAT_Master_ATxxxx.Beckhoff_AT1xxx.Beckhoff_AT2xxxEK1122.A_0032_AT2026_0250_0023.CC_Outputs.Current_setpoint_value_Ch[3] <-> CC Outputs/Current setpoint value Ch.4
//     PlcTask Outputs/GVL_iXlinker.EtherCAT_Master_ATxxxx.Beckhoff_AT1xxx.Beckhoff_AT2xxxEK1122.A_0032_AT2026_0250_0023.CC_Outputs.Current_setpoint_value_Ch[4] <-> CC Outputs/Current setpoint value Ch.5
//     PlcTask Outputs/GVL_iXlinker.EtherCAT_Master_ATxxxx.Beckhoff_AT1xxx.Beckhoff_AT2xxxEK1122.A_0032_AT2026_0250_0023.CC_Outputs.Current_setpoint_value_Ch[5] <-> CC Outputs/Current setpoint value Ch.6
//     PlcTask Outputs/GVL_iXlinker.EtherCAT_Master_ATxxxx.Beckhoff_AT1xxx.Beckhoff_AT2xxxEK1122.A_0032_AT2026_0250_0023.CC_Outputs.Current_setpoint_value_Ch[6] <-> CC Outputs/Current setpoint value Ch.7
//     PlcTask Outputs/GVL_iXlinker.EtherCAT_Master_ATxxxx.Beckhoff_AT1xxx.Beckhoff_AT2xxxEK1122.A_0032_AT2026_0250_0023.CC_Outputs.Current_setpoint_value_Ch[7] <-> CC Outputs/Current setpoint value Ch.8
//     PlcTask Outputs/GVL_iXlinker.EtherCAT_Master_ATxxxx.Beckhoff_AT1xxx.Beckhoff_AT2xxxEK1122.A_0032_AT2026_0250_0023.CC_Outputs.Current_setpoint_value_Ch[8] <-> CC Outputs/Current setpoint value Ch.9
//     PlcTask Outputs/GVL_iXlinker.EtherCAT_Master_ATxxxx.Beckhoff_AT1xxx.Beckhoff_AT2xxxEK1122.A_0032_AT2026_0250_0023.CC_Outputs.Current_setpoint_value_Ch[9] <-> CC Outputs/Current setpoint value Ch.10
//     PlcTask Outputs/GVL_iXlinker.EtherCAT_Master_ATxxxx.Beckhoff_AT1xxx.Beckhoff_AT2xxxEK1122.A_0032_AT2026_0250_0023.CC_Outputs.Current_setpoint_value_Ch[10] <-> CC Outputs/Current setpoint value Ch.11
//     PlcTask Outputs/GVL_iXlinker.EtherCAT_Master_ATxxxx.Beckhoff_AT1xxx.Beckhoff_AT2xxxEK1122.A_0032_AT2026_0250_0023.CC_Outputs.Current_setpoint_value_Ch[11] <-> CC Outputs/Current setpoint value Ch.12
//     PlcTask Outputs/GVL_iXlinker.EtherCAT_Master_ATxxxx.Beckhoff_AT1xxx.Beckhoff_AT2xxxEK1122.A_0032_AT2026_0250_0023.CC_Outputs.Current_setpoint_value_Ch[12] <-> CC Outputs/Current setpoint value Ch.13
//     PlcTask Outputs/GVL_iXlinker.EtherCAT_Master_ATxxxx.Beckhoff_AT1xxx.Beckhoff_AT2xxxEK1122.A_0032_AT2026_0250_0023.CC_Outputs.Current_setpoint_value_Ch[13] <-> CC Outputs/Current setpoint value Ch.14
//     PlcTask Outputs/GVL_iXlinker.EtherCAT_Master_ATxxxx.Beckhoff_AT1xxx.Beckhoff_AT2xxxEK1122.A_0032_AT2026_0250_0023.CC_Outputs.Current_setpoint_value_Ch[14] <-> CC Outputs/Current setpoint value Ch.15
//     PlcTask Inputs/GVL_iXlinker.EtherCAT_Master_ATxxxx.Beckhoff_AT1xxx.Beckhoff_AT2xxxEK1122.A_0032_AT2026_0250_0023.WcState.WcState <-> WcState/WcState
//     PlcTask Inputs/GVL_iXlinker.EtherCAT_Master_ATxxxx.Beckhoff_AT1xxx.Beckhoff_AT2xxxEK1122.A_0032_AT2026_0250_0023.WcState.InputToggle <-> WcState/InputToggle
//     PlcTask Inputs/GVL_iXlinker.EtherCAT_Master_ATxxxx.Beckhoff_AT1xxx.Beckhoff_AT2xxxEK1122.A_0032_AT2026_0250_0023.InfoData.AdsAddr <-> InfoData/AdsAddr
//     PlcTask Inputs/GVL_iXlinker.EtherCAT_Master_ATxxxx.Beckhoff_AT1xxx.Beckhoff_AT2xxxEK1122.A_0032_AT2026_0250_0023.InfoData.DcOutputShift <-> InfoData/DcOutputShift
//     PlcTask Inputs/GVL_iXlinker.EtherCAT_Master_ATxxxx.Beckhoff_AT1xxx.Beckhoff_AT2xxxEK1122.A_0032_AT2026_0250_0023.InfoData.DcInputShift <-> InfoData/DcInputShift
//     PlcTask Inputs/GVL_iXlinker.EtherCAT_Master_ATxxxx.Beckhoff_AT1xxx.Beckhoff_AT2xxxEK1122.A_0032_AT2026_0250_0023.InfoData.State <-> InfoData/State
//   PLC/PLC Instance <-> EtherCAT Master ATxxxx/Beckhoff AT1xxx/Beckhoff AT2xxxEK1122/A_0033(AT2040-0250-0018)
//     PlcTask Inputs/GVL_iXlinker.EtherCAT_Master_ATxxxx.Beckhoff_AT1xxx.Beckhoff_AT2xxxEK1122.A_0033_AT2040_0250_0018.CC_Inputs.Status <-> CC Inputs/Status
//     PlcTask Inputs/GVL_iXlinker.EtherCAT_Master_ATxxxx.Beckhoff_AT1xxx.Beckhoff_AT2xxxEK1122.A_0033_AT2040_0250_0018.CC_Inputs.Current_actual_value_Ch[0] <-> CC Inputs/Current actual value Ch.1
//     PlcTask Inputs/GVL_iXlinker.EtherCAT_Master_ATxxxx.Beckhoff_AT1xxx.Beckhoff_AT2xxxEK1122.A_0033_AT2040_0250_0018.CC_Inputs.Current_actual_value_Ch[1] <-> CC Inputs/Current actual value Ch.2
//     PlcTask Inputs/GVL_iXlinker.EtherCAT_Master_ATxxxx.Beckhoff_AT1xxx.Beckhoff_AT2xxxEK1122.A_0033_AT2040_0250_0018.CC_Inputs.Current_actual_value_Ch[2] <-> CC Inputs/Current actual value Ch.3
//     PlcTask Inputs/GVL_iXlinker.EtherCAT_Master_ATxxxx.Beckhoff_AT1xxx.Beckhoff_AT2xxxEK1122.A_0033_AT2040_0250_0018.CC_Inputs.Current_actual_value_Ch[3] <-> CC Inputs/Current actual value Ch.4
//     PlcTask Inputs/GVL_iXlinker.EtherCAT_Master_ATxxxx.Beckhoff_AT1xxx.Beckhoff_AT2xxxEK1122.A_0033_AT2040_0250_0018.CC_Inputs.Current_actual_value_Ch[4] <-> CC Inputs/Current actual value Ch.5
//     PlcTask Inputs/GVL_iXlinker.EtherCAT_Master_ATxxxx.Beckhoff_AT1xxx.Beckhoff_AT2xxxEK1122.A_0033_AT2040_0250_0018.CC_Inputs.Current_actual_value_Ch[5] <-> CC Inputs/Current actual value Ch.6
//     PlcTask Inputs/GVL_iXlinker.EtherCAT_Master_ATxxxx.Beckhoff_AT1xxx.Beckhoff_AT2xxxEK1122.A_0033_AT2040_0250_0018.CC_Inputs.Current_actual_value_Ch[6] <-> CC Inputs/Current actual value Ch.7
//     PlcTask Inputs/GVL_iXlinker.EtherCAT_Master_ATxxxx.Beckhoff_AT1xxx.Beckhoff_AT2xxxEK1122.A_0033_AT2040_0250_0018.CC_Inputs.Current_actual_value_Ch[7] <-> CC Inputs/Current actual value Ch.8
//     PlcTask Inputs/GVL_iXlinker.EtherCAT_Master_ATxxxx.Beckhoff_AT1xxx.Beckhoff_AT2xxxEK1122.A_0033_AT2040_0250_0018.CC_Inputs.Current_actual_value_Ch[8] <-> CC Inputs/Current actual value Ch.9
//     PlcTask Inputs/GVL_iXlinker.EtherCAT_Master_ATxxxx.Beckhoff_AT1xxx.Beckhoff_AT2xxxEK1122.A_0033_AT2040_0250_0018.CC_Inputs.Current_actual_value_Ch[9] <-> CC Inputs/Current actual value Ch.10
//     PlcTask Inputs/GVL_iXlinker.EtherCAT_Master_ATxxxx.Beckhoff_AT1xxx.Beckhoff_AT2xxxEK1122.A_0033_AT2040_0250_0018.CC_Inputs.Current_actual_value_Ch[10] <-> CC Inputs/Current actual value Ch.11
//     PlcTask Inputs/GVL_iXlinker.EtherCAT_Master_ATxxxx.Beckhoff_AT1xxx.Beckhoff_AT2xxxEK1122.A_0033_AT2040_0250_0018.CC_Inputs.Current_actual_value_Ch[11] <-> CC Inputs/Current actual value Ch.12
//     PlcTask Inputs/GVL_iXlinker.EtherCAT_Master_ATxxxx.Beckhoff_AT1xxx.Beckhoff_AT2xxxEK1122.A_0033_AT2040_0250_0018.CC_Inputs.Current_actual_value_Ch[12] <-> CC Inputs/Current actual value Ch.13
//     PlcTask Inputs/GVL_iXlinker.EtherCAT_Master_ATxxxx.Beckhoff_AT1xxx.Beckhoff_AT2xxxEK1122.A_0033_AT2040_0250_0018.CC_Inputs.Current_actual_value_Ch[13] <-> CC Inputs/Current actual value Ch.14
//     PlcTask Inputs/GVL_iXlinker.EtherCAT_Master_ATxxxx.Beckhoff_AT1xxx.Beckhoff_AT2xxxEK1122.A_0033_AT2040_0250_0018.CC_Inputs.Current_actual_value_Ch[14] <-> CC Inputs/Current actual value Ch.15
//     PlcTask Outputs/GVL_iXlinker.EtherCAT_Master_ATxxxx.Beckhoff_AT1xxx.Beckhoff_AT2xxxEK1122.A_0033_AT2040_0250_0018.CC_Outputs.Control <-> CC Outputs/Control
//     PlcTask Outputs/GVL_iXlinker.EtherCAT_Master_ATxxxx.Beckhoff_AT1xxx.Beckhoff_AT2xxxEK1122.A_0033_AT2040_0250_0018.CC_Outputs.Current_setpoint_value_Ch[0] <-> CC Outputs/Current setpoint value Ch.1
//     PlcTask Outputs/GVL_iXlinker.EtherCAT_Master_ATxxxx.Beckhoff_AT1xxx.Beckhoff_AT2xxxEK1122.A_0033_AT2040_0250_0018.CC_Outputs.Current_setpoint_value_Ch[1] <-> CC Outputs/Current setpoint value Ch.2
//     PlcTask Outputs/GVL_iXlinker.EtherCAT_Master_ATxxxx.Beckhoff_AT1xxx.Beckhoff_AT2xxxEK1122.A_0033_AT2040_0250_0018.CC_Outputs.Current_setpoint_value_Ch[2] <-> CC Outputs/Current setpoint value Ch.3
//     PlcTask Outputs/GVL_iXlinker.EtherCAT_Master_ATxxxx.Beckhoff_AT1xxx.Beckhoff_AT2xxxEK1122.A_0033_AT2040_0250_0018.CC_Outputs.Current_setpoint_value_Ch[3] <-> CC Outputs/Current setpoint value Ch.4
//     PlcTask Outputs/GVL_iXlinker.EtherCAT_Master_ATxxxx.Beckhoff_AT1xxx.Beckhoff_AT2xxxEK1122.A_0033_AT2040_0250_0018.CC_Outputs.Current_setpoint_value_Ch[4] <-> CC Outputs/Current setpoint value Ch.5
//     PlcTask Outputs/GVL_iXlinker.EtherCAT_Master_ATxxxx.Beckhoff_AT1xxx.Beckhoff_AT2xxxEK1122.A_0033_AT2040_0250_0018.CC_Outputs.Current_setpoint_value_Ch[5] <-> CC Outputs/Current setpoint value Ch.6
//     PlcTask Outputs/GVL_iXlinker.EtherCAT_Master_ATxxxx.Beckhoff_AT1xxx.Beckhoff_AT2xxxEK1122.A_0033_AT2040_0250_0018.CC_Outputs.Current_setpoint_value_Ch[6] <-> CC Outputs/Current setpoint value Ch.7
//     PlcTask Outputs/GVL_iXlinker.EtherCAT_Master_ATxxxx.Beckhoff_AT1xxx.Beckhoff_AT2xxxEK1122.A_0033_AT2040_0250_0018.CC_Outputs.Current_setpoint_value_Ch[7] <-> CC Outputs/Current setpoint value Ch.8
//     PlcTask Outputs/GVL_iXlinker.EtherCAT_Master_ATxxxx.Beckhoff_AT1xxx.Beckhoff_AT2xxxEK1122.A_0033_AT2040_0250_0018.CC_Outputs.Current_setpoint_value_Ch[8] <-> CC Outputs/Current setpoint value Ch.9
//     PlcTask Outputs/GVL_iXlinker.EtherCAT_Master_ATxxxx.Beckhoff_AT1xxx.Beckhoff_AT2xxxEK1122.A_0033_AT2040_0250_0018.CC_Outputs.Current_setpoint_value_Ch[9] <-> CC Outputs/Current setpoint value Ch.10
//     PlcTask Outputs/GVL_iXlinker.EtherCAT_Master_ATxxxx.Beckhoff_AT1xxx.Beckhoff_AT2xxxEK1122.A_0033_AT2040_0250_0018.CC_Outputs.Current_setpoint_value_Ch[10] <-> CC Outputs/Current setpoint value Ch.11
//     PlcTask Outputs/GVL_iXlinker.EtherCAT_Master_ATxxxx.Beckhoff_AT1xxx.Beckhoff_AT2xxxEK1122.A_0033_AT2040_0250_0018.CC_Outputs.Current_setpoint_value_Ch[11] <-> CC Outputs/Current setpoint value Ch.12
//     PlcTask Outputs/GVL_iXlinker.EtherCAT_Master_ATxxxx.Beckhoff_AT1xxx.Beckhoff_AT2xxxEK1122.A_0033_AT2040_0250_0018.CC_Outputs.Current_setpoint_value_Ch[12] <-> CC Outputs/Current setpoint value Ch.13
//     PlcTask Outputs/GVL_iXlinker.EtherCAT_Master_ATxxxx.Beckhoff_AT1xxx.Beckhoff_AT2xxxEK1122.A_0033_AT2040_0250_0018.CC_Outputs.Current_setpoint_value_Ch[13] <-> CC Outputs/Current setpoint value Ch.14
//     PlcTask Outputs/GVL_iXlinker.EtherCAT_Master_ATxxxx.Beckhoff_AT1xxx.Beckhoff_AT2xxxEK1122.A_0033_AT2040_0250_0018.CC_Outputs.Current_setpoint_value_Ch[14] <-> CC Outputs/Current setpoint value Ch.15
//     PlcTask Inputs/GVL_iXlinker.EtherCAT_Master_ATxxxx.Beckhoff_AT1xxx.Beckhoff_AT2xxxEK1122.A_0033_AT2040_0250_0018.WcState.WcState <-> WcState/WcState
//     PlcTask Inputs/GVL_iXlinker.EtherCAT_Master_ATxxxx.Beckhoff_AT1xxx.Beckhoff_AT2xxxEK1122.A_0033_AT2040_0250_0018.WcState.InputToggle <-> WcState/InputToggle
//     PlcTask Inputs/GVL_iXlinker.EtherCAT_Master_ATxxxx.Beckhoff_AT1xxx.Beckhoff_AT2xxxEK1122.A_0033_AT2040_0250_0018.InfoData.AdsAddr <-> InfoData/AdsAddr
//     PlcTask Inputs/GVL_iXlinker.EtherCAT_Master_ATxxxx.Beckhoff_AT1xxx.Beckhoff_AT2xxxEK1122.A_0033_AT2040_0250_0018.InfoData.DcOutputShift <-> InfoData/DcOutputShift
//     PlcTask Inputs/GVL_iXlinker.EtherCAT_Master_ATxxxx.Beckhoff_AT1xxx.Beckhoff_AT2xxxEK1122.A_0033_AT2040_0250_0018.InfoData.DcInputShift <-> InfoData/DcInputShift
//     PlcTask Inputs/GVL_iXlinker.EtherCAT_Master_ATxxxx.Beckhoff_AT1xxx.Beckhoff_AT2xxxEK1122.A_0033_AT2040_0250_0018.InfoData.State <-> InfoData/State
//   PLC/PLC Instance <-> EtherCAT Master ATxxxx/Beckhoff AT1xxx/Beckhoff AT2xxxEK1122/A_0034(AT2040-0250-0019)
//     PlcTask Inputs/GVL_iXlinker.EtherCAT_Master_ATxxxx.Beckhoff_AT1xxx.Beckhoff_AT2xxxEK1122.A_0034_AT2040_0250_0019.CC_Inputs.Status <-> CC Inputs/Status
//     PlcTask Inputs/GVL_iXlinker.EtherCAT_Master_ATxxxx.Beckhoff_AT1xxx.Beckhoff_AT2xxxEK1122.A_0034_AT2040_0250_0019.CC_Inputs.Current_actual_value_Ch[0] <-> CC Inputs/Current actual value Ch.1
//     PlcTask Inputs/GVL_iXlinker.EtherCAT_Master_ATxxxx.Beckhoff_AT1xxx.Beckhoff_AT2xxxEK1122.A_0034_AT2040_0250_0019.CC_Inputs.Current_actual_value_Ch[1] <-> CC Inputs/Current actual value Ch.2
//     PlcTask Inputs/GVL_iXlinker.EtherCAT_Master_ATxxxx.Beckhoff_AT1xxx.Beckhoff_AT2xxxEK1122.A_0034_AT2040_0250_0019.CC_Inputs.Current_actual_value_Ch[2] <-> CC Inputs/Current actual value Ch.3
//     PlcTask Inputs/GVL_iXlinker.EtherCAT_Master_ATxxxx.Beckhoff_AT1xxx.Beckhoff_AT2xxxEK1122.A_0034_AT2040_0250_0019.CC_Inputs.Current_actual_value_Ch[3] <-> CC Inputs/Current actual value Ch.4
//     PlcTask Inputs/GVL_iXlinker.EtherCAT_Master_ATxxxx.Beckhoff_AT1xxx.Beckhoff_AT2xxxEK1122.A_0034_AT2040_0250_0019.CC_Inputs.Current_actual_value_Ch[4] <-> CC Inputs/Current actual value Ch.5
//     PlcTask Inputs/GVL_iXlinker.EtherCAT_Master_ATxxxx.Beckhoff_AT1xxx.Beckhoff_AT2xxxEK1122.A_0034_AT2040_0250_0019.CC_Inputs.Current_actual_value_Ch[5] <-> CC Inputs/Current actual value Ch.6
//     PlcTask Inputs/GVL_iXlinker.EtherCAT_Master_ATxxxx.Beckhoff_AT1xxx.Beckhoff_AT2xxxEK1122.A_0034_AT2040_0250_0019.CC_Inputs.Current_actual_value_Ch[6] <-> CC Inputs/Current actual value Ch.7
//     PlcTask Inputs/GVL_iXlinker.EtherCAT_Master_ATxxxx.Beckhoff_AT1xxx.Beckhoff_AT2xxxEK1122.A_0034_AT2040_0250_0019.CC_Inputs.Current_actual_value_Ch[7] <-> CC Inputs/Current actual value Ch.8
//     PlcTask Inputs/GVL_iXlinker.EtherCAT_Master_ATxxxx.Beckhoff_AT1xxx.Beckhoff_AT2xxxEK1122.A_0034_AT2040_0250_0019.CC_Inputs.Current_actual_value_Ch[8] <-> CC Inputs/Current actual value Ch.9
//     PlcTask Inputs/GVL_iXlinker.EtherCAT_Master_ATxxxx.Beckhoff_AT1xxx.Beckhoff_AT2xxxEK1122.A_0034_AT2040_0250_0019.CC_Inputs.Current_actual_value_Ch[9] <-> CC Inputs/Current actual value Ch.10
//     PlcTask Inputs/GVL_iXlinker.EtherCAT_Master_ATxxxx.Beckhoff_AT1xxx.Beckhoff_AT2xxxEK1122.A_0034_AT2040_0250_0019.CC_Inputs.Current_actual_value_Ch[10] <-> CC Inputs/Current actual value Ch.11
//     PlcTask Inputs/GVL_iXlinker.EtherCAT_Master_ATxxxx.Beckhoff_AT1xxx.Beckhoff_AT2xxxEK1122.A_0034_AT2040_0250_0019.CC_Inputs.Current_actual_value_Ch[11] <-> CC Inputs/Current actual value Ch.12
//     PlcTask Inputs/GVL_iXlinker.EtherCAT_Master_ATxxxx.Beckhoff_AT1xxx.Beckhoff_AT2xxxEK1122.A_0034_AT2040_0250_0019.CC_Inputs.Current_actual_value_Ch[12] <-> CC Inputs/Current actual value Ch.13
//     PlcTask Inputs/GVL_iXlinker.EtherCAT_Master_ATxxxx.Beckhoff_AT1xxx.Beckhoff_AT2xxxEK1122.A_0034_AT2040_0250_0019.CC_Inputs.Current_actual_value_Ch[13] <-> CC Inputs/Current actual value Ch.14
//     PlcTask Inputs/GVL_iXlinker.EtherCAT_Master_ATxxxx.Beckhoff_AT1xxx.Beckhoff_AT2xxxEK1122.A_0034_AT2040_0250_0019.CC_Inputs.Current_actual_value_Ch[14] <-> CC Inputs/Current actual value Ch.15
//     PlcTask Outputs/GVL_iXlinker.EtherCAT_Master_ATxxxx.Beckhoff_AT1xxx.Beckhoff_AT2xxxEK1122.A_0034_AT2040_0250_0019.CC_Outputs.Control <-> CC Outputs/Control
//     PlcTask Outputs/GVL_iXlinker.EtherCAT_Master_ATxxxx.Beckhoff_AT1xxx.Beckhoff_AT2xxxEK1122.A_0034_AT2040_0250_0019.CC_Outputs.Current_setpoint_value_Ch[0] <-> CC Outputs/Current setpoint value Ch.1
//     PlcTask Outputs/GVL_iXlinker.EtherCAT_Master_ATxxxx.Beckhoff_AT1xxx.Beckhoff_AT2xxxEK1122.A_0034_AT2040_0250_0019.CC_Outputs.Current_setpoint_value_Ch[1] <-> CC Outputs/Current setpoint value Ch.2
//     PlcTask Outputs/GVL_iXlinker.EtherCAT_Master_ATxxxx.Beckhoff_AT1xxx.Beckhoff_AT2xxxEK1122.A_0034_AT2040_0250_0019.CC_Outputs.Current_setpoint_value_Ch[2] <-> CC Outputs/Current setpoint value Ch.3
//     PlcTask Outputs/GVL_iXlinker.EtherCAT_Master_ATxxxx.Beckhoff_AT1xxx.Beckhoff_AT2xxxEK1122.A_0034_AT2040_0250_0019.CC_Outputs.Current_setpoint_value_Ch[3] <-> CC Outputs/Current setpoint value Ch.4
//     PlcTask Outputs/GVL_iXlinker.EtherCAT_Master_ATxxxx.Beckhoff_AT1xxx.Beckhoff_AT2xxxEK1122.A_0034_AT2040_0250_0019.CC_Outputs.Current_setpoint_value_Ch[4] <-> CC Outputs/Current setpoint value Ch.5
//     PlcTask Outputs/GVL_iXlinker.EtherCAT_Master_ATxxxx.Beckhoff_AT1xxx.Beckhoff_AT2xxxEK1122.A_0034_AT2040_0250_0019.CC_Outputs.Current_setpoint_value_Ch[5] <-> CC Outputs/Current setpoint value Ch.6
//     PlcTask Outputs/GVL_iXlinker.EtherCAT_Master_ATxxxx.Beckhoff_AT1xxx.Beckhoff_AT2xxxEK1122.A_0034_AT2040_0250_0019.CC_Outputs.Current_setpoint_value_Ch[6] <-> CC Outputs/Current setpoint value Ch.7
//     PlcTask Outputs/GVL_iXlinker.EtherCAT_Master_ATxxxx.Beckhoff_AT1xxx.Beckhoff_AT2xxxEK1122.A_0034_AT2040_0250_0019.CC_Outputs.Current_setpoint_value_Ch[7] <-> CC Outputs/Current setpoint value Ch.8
//     PlcTask Outputs/GVL_iXlinker.EtherCAT_Master_ATxxxx.Beckhoff_AT1xxx.Beckhoff_AT2xxxEK1122.A_0034_AT2040_0250_0019.CC_Outputs.Current_setpoint_value_Ch[8] <-> CC Outputs/Current setpoint value Ch.9
//     PlcTask Outputs/GVL_iXlinker.EtherCAT_Master_ATxxxx.Beckhoff_AT1xxx.Beckhoff_AT2xxxEK1122.A_0034_AT2040_0250_0019.CC_Outputs.Current_setpoint_value_Ch[9] <-> CC Outputs/Current setpoint value Ch.10
//     PlcTask Outputs/GVL_iXlinker.EtherCAT_Master_ATxxxx.Beckhoff_AT1xxx.Beckhoff_AT2xxxEK1122.A_0034_AT2040_0250_0019.CC_Outputs.Current_setpoint_value_Ch[10] <-> CC Outputs/Current setpoint value Ch.11
//     PlcTask Outputs/GVL_iXlinker.EtherCAT_Master_ATxxxx.Beckhoff_AT1xxx.Beckhoff_AT2xxxEK1122.A_0034_AT2040_0250_0019.CC_Outputs.Current_setpoint_value_Ch[11] <-> CC Outputs/Current setpoint value Ch.12
//     PlcTask Outputs/GVL_iXlinker.EtherCAT_Master_ATxxxx.Beckhoff_AT1xxx.Beckhoff_AT2xxxEK1122.A_0034_AT2040_0250_0019.CC_Outputs.Current_setpoint_value_Ch[12] <-> CC Outputs/Current setpoint value Ch.13
//     PlcTask Outputs/GVL_iXlinker.EtherCAT_Master_ATxxxx.Beckhoff_AT1xxx.Beckhoff_AT2xxxEK1122.A_0034_AT2040_0250_0019.CC_Outputs.Current_setpoint_value_Ch[13] <-> CC Outputs/Current setpoint value Ch.14
//     PlcTask Outputs/GVL_iXlinker.EtherCAT_Master_ATxxxx.Beckhoff_AT1xxx.Beckhoff_AT2xxxEK1122.A_0034_AT2040_0250_0019.CC_Outputs.Current_setpoint_value_Ch[14] <-> CC Outputs/Current setpoint value Ch.15
//     PlcTask Inputs/GVL_iXlinker.EtherCAT_Master_ATxxxx.Beckhoff_AT1xxx.Beckhoff_AT2xxxEK1122.A_0034_AT2040_0250_0019.WcState.WcState <-> WcState/WcState
//     PlcTask Inputs/GVL_iXlinker.EtherCAT_Master_ATxxxx.Beckhoff_AT1xxx.Beckhoff_AT2xxxEK1122.A_0034_AT2040_0250_0019.WcState.InputToggle <-> WcState/InputToggle
//     PlcTask Inputs/GVL_iXlinker.EtherCAT_Master_ATxxxx.Beckhoff_AT1xxx.Beckhoff_AT2xxxEK1122.A_0034_AT2040_0250_0019.InfoData.AdsAddr <-> InfoData/AdsAddr
//     PlcTask Inputs/GVL_iXlinker.EtherCAT_Master_ATxxxx.Beckhoff_AT1xxx.Beckhoff_AT2xxxEK1122.A_0034_AT2040_0250_0019.InfoData.DcOutputShift <-> InfoData/DcOutputShift
//     PlcTask Inputs/GVL_iXlinker.EtherCAT_Master_ATxxxx.Beckhoff_AT1xxx.Beckhoff_AT2xxxEK1122.A_0034_AT2040_0250_0019.InfoData.DcInputShift <-> InfoData/DcInputShift
//     PlcTask Inputs/GVL_iXlinker.EtherCAT_Master_ATxxxx.Beckhoff_AT1xxx.Beckhoff_AT2xxxEK1122.A_0034_AT2040_0250_0019.InfoData.State <-> InfoData/State
//   PLC/PLC Instance <-> EtherCAT Master ATxxxx/Beckhoff AT1xxx/Beckhoff AT2xxxEK1122/A_0035(AT2040-0250-0020)
//     PlcTask Inputs/GVL_iXlinker.EtherCAT_Master_ATxxxx.Beckhoff_AT1xxx.Beckhoff_AT2xxxEK1122.A_0035_AT2040_0250_0020.CC_Inputs.Status <-> CC Inputs/Status
//     PlcTask Inputs/GVL_iXlinker.EtherCAT_Master_ATxxxx.Beckhoff_AT1xxx.Beckhoff_AT2xxxEK1122.A_0035_AT2040_0250_0020.CC_Inputs.Current_actual_value_Ch[0] <-> CC Inputs/Current actual value Ch.1
//     PlcTask Inputs/GVL_iXlinker.EtherCAT_Master_ATxxxx.Beckhoff_AT1xxx.Beckhoff_AT2xxxEK1122.A_0035_AT2040_0250_0020.CC_Inputs.Current_actual_value_Ch[1] <-> CC Inputs/Current actual value Ch.2
//     PlcTask Inputs/GVL_iXlinker.EtherCAT_Master_ATxxxx.Beckhoff_AT1xxx.Beckhoff_AT2xxxEK1122.A_0035_AT2040_0250_0020.CC_Inputs.Current_actual_value_Ch[2] <-> CC Inputs/Current actual value Ch.3
//     PlcTask Inputs/GVL_iXlinker.EtherCAT_Master_ATxxxx.Beckhoff_AT1xxx.Beckhoff_AT2xxxEK1122.A_0035_AT2040_0250_0020.CC_Inputs.Current_actual_value_Ch[3] <-> CC Inputs/Current actual value Ch.4
//     PlcTask Inputs/GVL_iXlinker.EtherCAT_Master_ATxxxx.Beckhoff_AT1xxx.Beckhoff_AT2xxxEK1122.A_0035_AT2040_0250_0020.CC_Inputs.Current_actual_value_Ch[4] <-> CC Inputs/Current actual value Ch.5
//     PlcTask Inputs/GVL_iXlinker.EtherCAT_Master_ATxxxx.Beckhoff_AT1xxx.Beckhoff_AT2xxxEK1122.A_0035_AT2040_0250_0020.CC_Inputs.Current_actual_value_Ch[5] <-> CC Inputs/Current actual value Ch.6
//     PlcTask Inputs/GVL_iXlinker.EtherCAT_Master_ATxxxx.Beckhoff_AT1xxx.Beckhoff_AT2xxxEK1122.A_0035_AT2040_0250_0020.CC_Inputs.Current_actual_value_Ch[6] <-> CC Inputs/Current actual value Ch.7
//     PlcTask Inputs/GVL_iXlinker.EtherCAT_Master_ATxxxx.Beckhoff_AT1xxx.Beckhoff_AT2xxxEK1122.A_0035_AT2040_0250_0020.CC_Inputs.Current_actual_value_Ch[7] <-> CC Inputs/Current actual value Ch.8
//     PlcTask Inputs/GVL_iXlinker.EtherCAT_Master_ATxxxx.Beckhoff_AT1xxx.Beckhoff_AT2xxxEK1122.A_0035_AT2040_0250_0020.CC_Inputs.Current_actual_value_Ch[8] <-> CC Inputs/Current actual value Ch.9
//     PlcTask Inputs/GVL_iXlinker.EtherCAT_Master_ATxxxx.Beckhoff_AT1xxx.Beckhoff_AT2xxxEK1122.A_0035_AT2040_0250_0020.CC_Inputs.Current_actual_value_Ch[9] <-> CC Inputs/Current actual value Ch.10
//     PlcTask Inputs/GVL_iXlinker.EtherCAT_Master_ATxxxx.Beckhoff_AT1xxx.Beckhoff_AT2xxxEK1122.A_0035_AT2040_0250_0020.CC_Inputs.Current_actual_value_Ch[10] <-> CC Inputs/Current actual value Ch.11
//     PlcTask Inputs/GVL_iXlinker.EtherCAT_Master_ATxxxx.Beckhoff_AT1xxx.Beckhoff_AT2xxxEK1122.A_0035_AT2040_0250_0020.CC_Inputs.Current_actual_value_Ch[11] <-> CC Inputs/Current actual value Ch.12
//     PlcTask Inputs/GVL_iXlinker.EtherCAT_Master_ATxxxx.Beckhoff_AT1xxx.Beckhoff_AT2xxxEK1122.A_0035_AT2040_0250_0020.CC_Inputs.Current_actual_value_Ch[12] <-> CC Inputs/Current actual value Ch.13
//     PlcTask Inputs/GVL_iXlinker.EtherCAT_Master_ATxxxx.Beckhoff_AT1xxx.Beckhoff_AT2xxxEK1122.A_0035_AT2040_0250_0020.CC_Inputs.Current_actual_value_Ch[13] <-> CC Inputs/Current actual value Ch.14
//     PlcTask Inputs/GVL_iXlinker.EtherCAT_Master_ATxxxx.Beckhoff_AT1xxx.Beckhoff_AT2xxxEK1122.A_0035_AT2040_0250_0020.CC_Inputs.Current_actual_value_Ch[14] <-> CC Inputs/Current actual value Ch.15
//     PlcTask Outputs/GVL_iXlinker.EtherCAT_Master_ATxxxx.Beckhoff_AT1xxx.Beckhoff_AT2xxxEK1122.A_0035_AT2040_0250_0020.CC_Outputs.Control <-> CC Outputs/Control
//     PlcTask Outputs/GVL_iXlinker.EtherCAT_Master_ATxxxx.Beckhoff_AT1xxx.Beckhoff_AT2xxxEK1122.A_0035_AT2040_0250_0020.CC_Outputs.Current_setpoint_value_Ch[0] <-> CC Outputs/Current setpoint value Ch.1
//     PlcTask Outputs/GVL_iXlinker.EtherCAT_Master_ATxxxx.Beckhoff_AT1xxx.Beckhoff_AT2xxxEK1122.A_0035_AT2040_0250_0020.CC_Outputs.Current_setpoint_value_Ch[1] <-> CC Outputs/Current setpoint value Ch.2
//     PlcTask Outputs/GVL_iXlinker.EtherCAT_Master_ATxxxx.Beckhoff_AT1xxx.Beckhoff_AT2xxxEK1122.A_0035_AT2040_0250_0020.CC_Outputs.Current_setpoint_value_Ch[2] <-> CC Outputs/Current setpoint value Ch.3
//     PlcTask Outputs/GVL_iXlinker.EtherCAT_Master_ATxxxx.Beckhoff_AT1xxx.Beckhoff_AT2xxxEK1122.A_0035_AT2040_0250_0020.CC_Outputs.Current_setpoint_value_Ch[3] <-> CC Outputs/Current setpoint value Ch.4
//     PlcTask Outputs/GVL_iXlinker.EtherCAT_Master_ATxxxx.Beckhoff_AT1xxx.Beckhoff_AT2xxxEK1122.A_0035_AT2040_0250_0020.CC_Outputs.Current_setpoint_value_Ch[4] <-> CC Outputs/Current setpoint value Ch.5
//     PlcTask Outputs/GVL_iXlinker.EtherCAT_Master_ATxxxx.Beckhoff_AT1xxx.Beckhoff_AT2xxxEK1122.A_0035_AT2040_0250_0020.CC_Outputs.Current_setpoint_value_Ch[5] <-> CC Outputs/Current setpoint value Ch.6
//     PlcTask Outputs/GVL_iXlinker.EtherCAT_Master_ATxxxx.Beckhoff_AT1xxx.Beckhoff_AT2xxxEK1122.A_0035_AT2040_0250_0020.CC_Outputs.Current_setpoint_value_Ch[6] <-> CC Outputs/Current setpoint value Ch.7
//     PlcTask Outputs/GVL_iXlinker.EtherCAT_Master_ATxxxx.Beckhoff_AT1xxx.Beckhoff_AT2xxxEK1122.A_0035_AT2040_0250_0020.CC_Outputs.Current_setpoint_value_Ch[7] <-> CC Outputs/Current setpoint value Ch.8
//     PlcTask Outputs/GVL_iXlinker.EtherCAT_Master_ATxxxx.Beckhoff_AT1xxx.Beckhoff_AT2xxxEK1122.A_0035_AT2040_0250_0020.CC_Outputs.Current_setpoint_value_Ch[8] <-> CC Outputs/Current setpoint value Ch.9
//     PlcTask Outputs/GVL_iXlinker.EtherCAT_Master_ATxxxx.Beckhoff_AT1xxx.Beckhoff_AT2xxxEK1122.A_0035_AT2040_0250_0020.CC_Outputs.Current_setpoint_value_Ch[9] <-> CC Outputs/Current setpoint value Ch.10
//     PlcTask Outputs/GVL_iXlinker.EtherCAT_Master_ATxxxx.Beckhoff_AT1xxx.Beckhoff_AT2xxxEK1122.A_0035_AT2040_0250_0020.CC_Outputs.Current_setpoint_value_Ch[10] <-> CC Outputs/Current setpoint value Ch.11
//     PlcTask Outputs/GVL_iXlinker.EtherCAT_Master_ATxxxx.Beckhoff_AT1xxx.Beckhoff_AT2xxxEK1122.A_0035_AT2040_0250_0020.CC_Outputs.Current_setpoint_value_Ch[11] <-> CC Outputs/Current setpoint value Ch.12
//     PlcTask Outputs/GVL_iXlinker.EtherCAT_Master_ATxxxx.Beckhoff_AT1xxx.Beckhoff_AT2xxxEK1122.A_0035_AT2040_0250_0020.CC_Outputs.Current_setpoint_value_Ch[12] <-> CC Outputs/Current setpoint value Ch.13
//     PlcTask Outputs/GVL_iXlinker.EtherCAT_Master_ATxxxx.Beckhoff_AT1xxx.Beckhoff_AT2xxxEK1122.A_0035_AT2040_0250_0020.CC_Outputs.Current_setpoint_value_Ch[13] <-> CC Outputs/Current setpoint value Ch.14
//     PlcTask Outputs/GVL_iXlinker.EtherCAT_Master_ATxxxx.Beckhoff_AT1xxx.Beckhoff_AT2xxxEK1122.A_0035_AT2040_0250_0020.CC_Outputs.Current_setpoint_value_Ch[14] <-> CC Outputs/Current setpoint value Ch.15
//     PlcTask Inputs/GVL_iXlinker.EtherCAT_Master_ATxxxx.Beckhoff_AT1xxx.Beckhoff_AT2xxxEK1122.A_0035_AT2040_0250_0020.WcState.WcState <-> WcState/WcState
//     PlcTask Inputs/GVL_iXlinker.EtherCAT_Master_ATxxxx.Beckhoff_AT1xxx.Beckhoff_AT2xxxEK1122.A_0035_AT2040_0250_0020.WcState.InputToggle <-> WcState/InputToggle
//     PlcTask Inputs/GVL_iXlinker.EtherCAT_Master_ATxxxx.Beckhoff_AT1xxx.Beckhoff_AT2xxxEK1122.A_0035_AT2040_0250_0020.InfoData.AdsAddr <-> InfoData/AdsAddr
//     PlcTask Inputs/GVL_iXlinker.EtherCAT_Master_ATxxxx.Beckhoff_AT1xxx.Beckhoff_AT2xxxEK1122.A_0035_AT2040_0250_0020.InfoData.DcOutputShift <-> InfoData/DcOutputShift
//     PlcTask Inputs/GVL_iXlinker.EtherCAT_Master_ATxxxx.Beckhoff_AT1xxx.Beckhoff_AT2xxxEK1122.A_0035_AT2040_0250_0020.InfoData.DcInputShift <-> InfoData/DcInputShift
//     PlcTask Inputs/GVL_iXlinker.EtherCAT_Master_ATxxxx.Beckhoff_AT1xxx.Beckhoff_AT2xxxEK1122.A_0035_AT2040_0250_0020.InfoData.State <-> InfoData/State
//   PLC/PLC Instance <-> EtherCAT Master ATxxxx/Beckhoff AT1xxx/Beckhoff AT2xxxEK1122/A_0036(AT2040-0250-0021)
//     PlcTask Inputs/GVL_iXlinker.EtherCAT_Master_ATxxxx.Beckhoff_AT1xxx.Beckhoff_AT2xxxEK1122.A_0036_AT2040_0250_0021.CC_Inputs.Status <-> CC Inputs/Status
//     PlcTask Inputs/GVL_iXlinker.EtherCAT_Master_ATxxxx.Beckhoff_AT1xxx.Beckhoff_AT2xxxEK1122.A_0036_AT2040_0250_0021.CC_Inputs.Current_actual_value_Ch[0] <-> CC Inputs/Current actual value Ch.1
//     PlcTask Inputs/GVL_iXlinker.EtherCAT_Master_ATxxxx.Beckhoff_AT1xxx.Beckhoff_AT2xxxEK1122.A_0036_AT2040_0250_0021.CC_Inputs.Current_actual_value_Ch[1] <-> CC Inputs/Current actual value Ch.2
//     PlcTask Inputs/GVL_iXlinker.EtherCAT_Master_ATxxxx.Beckhoff_AT1xxx.Beckhoff_AT2xxxEK1122.A_0036_AT2040_0250_0021.CC_Inputs.Current_actual_value_Ch[2] <-> CC Inputs/Current actual value Ch.3
//     PlcTask Inputs/GVL_iXlinker.EtherCAT_Master_ATxxxx.Beckhoff_AT1xxx.Beckhoff_AT2xxxEK1122.A_0036_AT2040_0250_0021.CC_Inputs.Current_actual_value_Ch[3] <-> CC Inputs/Current actual value Ch.4
//     PlcTask Inputs/GVL_iXlinker.EtherCAT_Master_ATxxxx.Beckhoff_AT1xxx.Beckhoff_AT2xxxEK1122.A_0036_AT2040_0250_0021.CC_Inputs.Current_actual_value_Ch[4] <-> CC Inputs/Current actual value Ch.5
//     PlcTask Inputs/GVL_iXlinker.EtherCAT_Master_ATxxxx.Beckhoff_AT1xxx.Beckhoff_AT2xxxEK1122.A_0036_AT2040_0250_0021.CC_Inputs.Current_actual_value_Ch[5] <-> CC Inputs/Current actual value Ch.6
//     PlcTask Inputs/GVL_iXlinker.EtherCAT_Master_ATxxxx.Beckhoff_AT1xxx.Beckhoff_AT2xxxEK1122.A_0036_AT2040_0250_0021.CC_Inputs.Current_actual_value_Ch[6] <-> CC Inputs/Current actual value Ch.7
//     PlcTask Inputs/GVL_iXlinker.EtherCAT_Master_ATxxxx.Beckhoff_AT1xxx.Beckhoff_AT2xxxEK1122.A_0036_AT2040_0250_0021.CC_Inputs.Current_actual_value_Ch[7] <-> CC Inputs/Current actual value Ch.8
//     PlcTask Inputs/GVL_iXlinker.EtherCAT_Master_ATxxxx.Beckhoff_AT1xxx.Beckhoff_AT2xxxEK1122.A_0036_AT2040_0250_0021.CC_Inputs.Current_actual_value_Ch[8] <-> CC Inputs/Current actual value Ch.9
//     PlcTask Inputs/GVL_iXlinker.EtherCAT_Master_ATxxxx.Beckhoff_AT1xxx.Beckhoff_AT2xxxEK1122.A_0036_AT2040_0250_0021.CC_Inputs.Current_actual_value_Ch[9] <-> CC Inputs/Current actual value Ch.10
//     PlcTask Inputs/GVL_iXlinker.EtherCAT_Master_ATxxxx.Beckhoff_AT1xxx.Beckhoff_AT2xxxEK1122.A_0036_AT2040_0250_0021.CC_Inputs.Current_actual_value_Ch[10] <-> CC Inputs/Current actual value Ch.11
//     PlcTask Inputs/GVL_iXlinker.EtherCAT_Master_ATxxxx.Beckhoff_AT1xxx.Beckhoff_AT2xxxEK1122.A_0036_AT2040_0250_0021.CC_Inputs.Current_actual_value_Ch[11] <-> CC Inputs/Current actual value Ch.12
//     PlcTask Inputs/GVL_iXlinker.EtherCAT_Master_ATxxxx.Beckhoff_AT1xxx.Beckhoff_AT2xxxEK1122.A_0036_AT2040_0250_0021.CC_Inputs.Current_actual_value_Ch[12] <-> CC Inputs/Current actual value Ch.13
//     PlcTask Inputs/GVL_iXlinker.EtherCAT_Master_ATxxxx.Beckhoff_AT1xxx.Beckhoff_AT2xxxEK1122.A_0036_AT2040_0250_0021.CC_Inputs.Current_actual_value_Ch[13] <-> CC Inputs/Current actual value Ch.14
//     PlcTask Inputs/GVL_iXlinker.EtherCAT_Master_ATxxxx.Beckhoff_AT1xxx.Beckhoff_AT2xxxEK1122.A_0036_AT2040_0250_0021.CC_Inputs.Current_actual_value_Ch[14] <-> CC Inputs/Current actual value Ch.15
//     PlcTask Outputs/GVL_iXlinker.EtherCAT_Master_ATxxxx.Beckhoff_AT1xxx.Beckhoff_AT2xxxEK1122.A_0036_AT2040_0250_0021.CC_Outputs.Control <-> CC Outputs/Control
//     PlcTask Outputs/GVL_iXlinker.EtherCAT_Master_ATxxxx.Beckhoff_AT1xxx.Beckhoff_AT2xxxEK1122.A_0036_AT2040_0250_0021.CC_Outputs.Current_setpoint_value_Ch[0] <-> CC Outputs/Current setpoint value Ch.1
//     PlcTask Outputs/GVL_iXlinker.EtherCAT_Master_ATxxxx.Beckhoff_AT1xxx.Beckhoff_AT2xxxEK1122.A_0036_AT2040_0250_0021.CC_Outputs.Current_setpoint_value_Ch[1] <-> CC Outputs/Current setpoint value Ch.2
//     PlcTask Outputs/GVL_iXlinker.EtherCAT_Master_ATxxxx.Beckhoff_AT1xxx.Beckhoff_AT2xxxEK1122.A_0036_AT2040_0250_0021.CC_Outputs.Current_setpoint_value_Ch[2] <-> CC Outputs/Current setpoint value Ch.3
//     PlcTask Outputs/GVL_iXlinker.EtherCAT_Master_ATxxxx.Beckhoff_AT1xxx.Beckhoff_AT2xxxEK1122.A_0036_AT2040_0250_0021.CC_Outputs.Current_setpoint_value_Ch[3] <-> CC Outputs/Current setpoint value Ch.4
//     PlcTask Outputs/GVL_iXlinker.EtherCAT_Master_ATxxxx.Beckhoff_AT1xxx.Beckhoff_AT2xxxEK1122.A_0036_AT2040_0250_0021.CC_Outputs.Current_setpoint_value_Ch[4] <-> CC Outputs/Current setpoint value Ch.5
//     PlcTask Outputs/GVL_iXlinker.EtherCAT_Master_ATxxxx.Beckhoff_AT1xxx.Beckhoff_AT2xxxEK1122.A_0036_AT2040_0250_0021.CC_Outputs.Current_setpoint_value_Ch[5] <-> CC Outputs/Current setpoint value Ch.6
//     PlcTask Outputs/GVL_iXlinker.EtherCAT_Master_ATxxxx.Beckhoff_AT1xxx.Beckhoff_AT2xxxEK1122.A_0036_AT2040_0250_0021.CC_Outputs.Current_setpoint_value_Ch[6] <-> CC Outputs/Current setpoint value Ch.7
//     PlcTask Outputs/GVL_iXlinker.EtherCAT_Master_ATxxxx.Beckhoff_AT1xxx.Beckhoff_AT2xxxEK1122.A_0036_AT2040_0250_0021.CC_Outputs.Current_setpoint_value_Ch[7] <-> CC Outputs/Current setpoint value Ch.8
//     PlcTask Outputs/GVL_iXlinker.EtherCAT_Master_ATxxxx.Beckhoff_AT1xxx.Beckhoff_AT2xxxEK1122.A_0036_AT2040_0250_0021.CC_Outputs.Current_setpoint_value_Ch[8] <-> CC Outputs/Current setpoint value Ch.9
//     PlcTask Outputs/GVL_iXlinker.EtherCAT_Master_ATxxxx.Beckhoff_AT1xxx.Beckhoff_AT2xxxEK1122.A_0036_AT2040_0250_0021.CC_Outputs.Current_setpoint_value_Ch[9] <-> CC Outputs/Current setpoint value Ch.10
//     PlcTask Outputs/GVL_iXlinker.EtherCAT_Master_ATxxxx.Beckhoff_AT1xxx.Beckhoff_AT2xxxEK1122.A_0036_AT2040_0250_0021.CC_Outputs.Current_setpoint_value_Ch[10] <-> CC Outputs/Current setpoint value Ch.11
//     PlcTask Outputs/GVL_iXlinker.EtherCAT_Master_ATxxxx.Beckhoff_AT1xxx.Beckhoff_AT2xxxEK1122.A_0036_AT2040_0250_0021.CC_Outputs.Current_setpoint_value_Ch[11] <-> CC Outputs/Current setpoint value Ch.12
//     PlcTask Outputs/GVL_iXlinker.EtherCAT_Master_ATxxxx.Beckhoff_AT1xxx.Beckhoff_AT2xxxEK1122.A_0036_AT2040_0250_0021.CC_Outputs.Current_setpoint_value_Ch[12] <-> CC Outputs/Current setpoint value Ch.13
//     PlcTask Outputs/GVL_iXlinker.EtherCAT_Master_ATxxxx.Beckhoff_AT1xxx.Beckhoff_AT2xxxEK1122.A_0036_AT2040_0250_0021.CC_Outputs.Current_setpoint_value_Ch[13] <-> CC Outputs/Current setpoint value Ch.14
//     PlcTask Outputs/GVL_iXlinker.EtherCAT_Master_ATxxxx.Beckhoff_AT1xxx.Beckhoff_AT2xxxEK1122.A_0036_AT2040_0250_0021.CC_Outputs.Current_setpoint_value_Ch[14] <-> CC Outputs/Current setpoint value Ch.15
